C01810=1081.766,322.523,409.402,175.975,26.438,154.460
C01811=1081.760,322.276,409.435,175.972,26.433,154.460
C01812=1081.754,322.027,409.468,175.969,26.429,154.459
C01813=1081.748,321.780,409.500,175.966,26.425,154.458
C01814=1081.742,321.532,409.533,175.963,26.420,154.458
C01815=1081.737,321.283,409.566,175.960,26.416,154.457
C01816=1081.731,321.037,409.598,175.957,26.412,154.457
C01817=1081.725,320.789,409.631,175.954,26.407,154.456
C01818=1081.717,320.468,409.673,175.950,26.402,154.455
C01819=1081.710,320.149,409.715,175.946,26.396,154.454
C01820=1081.702,319.829,409.757,175.943,26.390,154.453
C01821=1081.694,319.509,409.799,175.939,26.385,154.452
C01822=1081.689,319.262,409.831,175.936,26.380,154.452
C01823=1081.684,319.013,409.864,175.933,26.376,154.451
C01824=1081.677,318.766,409.897,175.930,26.372,154.450
C01825=1081.671,318.517,409.929,175.927,26.367,154.450
C01826=1081.666,318.270,409.962,175.924,26.363,154.449
C01827=1081.660,318.022,409.994,175.921,26.359,154.449
C01828=1081.654,317.774,410.026,175.918,26.355,154.448
C01829=1081.648,317.526,410.058,175.915,26.350,154.447
C01830=1081.640,317.181,410.104,175.911,26.344,154.446
C01831=1081.633,316.834,410.149,175.906,26.338,154.445
C01832=1081.625,316.489,410.194,175.903,26.333,154.445
C01833=1081.616,316.143,410.239,175.898,26.326,154.444
C01834=1081.611,315.895,410.271,175.895,26.322,154.443
C01835=1081.605,315.647,410.303,175.892,26.317,154.442
C01836=1081.599,315.399,410.335,175.890,26.314,154.442
C01837=1081.594,315.151,410.368,175.887,26.309,154.441
C01838=1081.588,314.903,410.400,175.884,26.305,154.440
C01839=1081.582,314.655,410.432,175.881,26.301,154.440
C01840=1081.576,314.407,410.464,175.878,26.296,154.439
C01841=1081.570,314.160,410.496,175.875,26.293,154.439
C01842=1081.564,313.912,410.528,175.872,26.288,154.438
C01843=1081.558,313.664,410.560,175.869,26.284,154.437
C01844=1081.552,313.416,410.592,175.866,26.280,154.437
C01845=1081.546,313.168,410.624,175.862,26.276,154.436
C01846=1081.540,312.920,410.656,175.859,26.272,154.436
C01847=1081.534,312.672,410.687,175.857,26.268,154.435
C01848=1081.528,312.424,410.719,175.854,26.264,154.434
C01849=1081.522,312.177,410.751,175.851,26.259,154.434
C01850=1081.516,311.929,410.783,175.848,26.256,154.433
C01851=1081.510,311.681,410.815,175.845,26.251,154.433
C01852=1081.504,311.433,410.847,175.842,26.247,154.432
C01853=1081.498,311.185,410.879,175.839,26.243,154.431
C01854=1081.492,310.937,410.910,175.836,26.239,154.431
C01855=1081.486,310.690,410.942,175.833,26.235,154.430
C01856=1081.480,310.442,410.973,175.831,26.231,154.430
C01857=1081.474,310.194,411.005,175.828,26.227,154.429
C01858=1081.468,309.946,411.037,175.824,26.223,154.428
C01859=1081.463,309.698,411.068,175.821,26.219,154.428
C01860=1081.457,309.450,411.100,175.818,26.215,154.427
C01861=1081.451,309.202,411.131,175.815,26.210,154.427
C01862=1081.445,308.954,411.163,175.812,26.207,154.426
C01863=1081.438,308.706,411.195,175.809,26.202,154.425
C01864=1081.433,308.458,411.227,175.807,26.199,154.425
C01865=1081.427,308.210,411.259,175.804,26.194,154.424
C01866=1081.421,307.962,411.289,175.801,26.190,154.424
C01867=1081.415,307.714,411.321,175.798,26.186,154.423
C01868=1081.410,307.467,411.353,175.795,26.182,154.423
C01869=1081.403,307.219,411.384,175.792,26.178,154.422
C01870=1081.398,306.971,411.416,175.789,26.174,154.421
C01871=1081.392,306.722,411.447,175.787,26.170,154.421
C01872=1081.386,306.475,411.478,175.784,26.166,154.420
C01873=1081.380,306.227,411.510,175.780,26.162,154.420
C01874=1081.375,305.980,411.542,175.777,26.158,154.419
C01875=1081.369,305.732,411.572,175.774,26.154,154.419
C01876=1081.363,305.483,411.604,175.771,26.150,154.418
C01877=1081.357,305.236,411.635,175.768,26.146,154.417
C01878=1081.351,304.987,411.667,175.766,26.142,154.417
C01879=1081.346,304.740,411.698,175.763,26.138,154.416
C01880=1081.339,304.491,411.729,175.760,26.134,154.416
C01881=1081.334,304.244,411.761,175.757,26.130,154.415
C01882=1081.324,303.829,411.813,175.752,26.123,154.414
C01883=1081.314,303.414,411.865,175.747,26.116,154.413
C01884=1081.305,302.999,411.918,175.743,26.109,154.412
C01885=1081.295,302.584,411.970,175.738,26.103,154.411
C01886=1081.289,302.336,412.000,175.735,26.099,154.411
C01887=1081.284,302.088,412.032,175.732,26.095,154.410
C01888=1081.278,301.840,412.063,175.729,26.091,154.409
C01889=1081.272,301.592,412.094,175.726,26.086,154.409
C01890=1081.267,301.344,412.125,175.724,26.083,154.408
C01891=1081.261,301.096,412.156,175.721,26.079,154.408
C01892=1081.255,300.848,412.188,175.718,26.075,154.407
C01893=1081.249,300.600,412.218,175.715,26.071,154.407
C01894=1081.244,300.352,412.249,175.711,26.067,154.406
C01895=1081.238,300.105,412.280,175.709,26.063,154.405
C01896=1081.232,299.856,412.311,175.706,26.059,154.405
C01897=1081.226,299.608,412.342,175.703,26.054,154.404
C01898=1081.221,299.361,412.373,175.700,26.051,154.404
C01899=1081.215,299.113,412.404,175.697,26.047,154.403
C01900=1081.209,298.864,412.435,175.695,26.043,154.402
C01901=1081.203,298.617,412.466,175.692,26.039,154.402
C01902=1081.198,298.369,412.497,175.689,26.035,154.401
C01903=1081.192,298.121,412.528,175.686,26.030,154.401
C01904=1081.187,297.873,412.558,175.684,26.027,154.400
C01905=1081.181,297.624,412.589,175.681,26.023,154.400
C01906=1081.175,297.376,412.620,175.678,26.019,154.399
C01907=1081.170,297.129,412.651,175.674,26.015,154.399
C01908=1081.163,296.880,412.682,175.671,26.011,154.398
C01909=1081.157,296.633,412.712,175.669,26.007,154.397
C01910=1081.152,296.384,412.743,175.666,26.003,154.397
C01911=1081.147,296.137,412.774,175.663,25.999,154.396
C01912=1081.141,295.889,412.804,175.660,25.996,154.396
C01913=1081.134,295.640,412.835,175.658,25.992,154.395
C01914=1081.129,295.392,412.865,175.655,25.988,154.395
C01915=1081.123,295.144,412.896,175.652,25.984,154.394
C01916=1081.118,294.896,412.926,175.649,25.980,154.394
C01917=1081.111,294.648,412.957,175.647,25.976,154.393
C01918=1081.105,294.400,412.987,175.643,25.972,154.393
C01919=1081.100,294.152,413.018,175.640,25.968,154.392
C01920=1081.094,293.904,413.048,175.637,25.965,154.392
C01921=1081.088,293.657,413.078,175.635,25.961,154.391
C01922=1081.082,293.408,413.110,175.632,25.957,154.391
C01923=1081.076,293.160,413.140,175.629,25.953,154.390
C01924=1081.071,292.912,413.170,175.627,25.950,154.389
C01925=1081.065,292.664,413.201,175.624,25.946,154.389
C01926=1081.059,292.417,413.231,175.621,25.942,154.388
C01927=1081.053,292.168,413.261,175.618,25.938,154.388
C01928=1081.047,291.920,413.291,175.615,25.934,154.387
C01929=1081.041,291.672,413.322,175.612,25.930,154.387
C01930=1081.035,291.424,413.352,175.609,25.927,154.386
C01931=1081.030,291.176,413.382,175.606,25.922,154.386
C01932=1081.024,290.928,413.412,175.604,25.919,154.385
C01933=1081.018,290.680,413.442,175.601,25.915,154.385
C01934=1081.009,290.279,413.491,175.596,25.909,154.384
C01935=1081.000,289.878,413.541,175.592,25.902,154.383
C01936=1080.990,289.478,413.589,175.587,25.896,154.382
C01937=1080.981,289.076,413.638,175.583,25.890,154.381
C01938=1080.975,288.829,413.668,175.580,25.886,154.381
C01939=1080.970,288.580,413.698,175.578,25.883,154.380
C01940=1080.964,288.332,413.728,175.574,25.879,154.380
C01941=1080.957,288.084,413.758,175.571,25.875,154.379
C01942=1080.951,287.836,413.788,175.569,25.872,154.379
C01943=1080.946,287.588,413.818,175.566,25.868,154.378
C01944=1080.940,287.339,413.848,175.563,25.864,154.378
C01945=1080.934,287.092,413.878,175.561,25.860,154.377
C01946=1080.929,286.843,413.908,175.558,25.857,154.377
C01947=1080.923,286.595,413.938,175.555,25.853,154.376
C01948=1080.917,286.347,413.967,175.553,25.849,154.376
C01949=1080.911,286.099,413.998,175.549,25.845,154.375
C01950=1080.905,285.851,414.027,175.546,25.842,154.375
C01951=1080.900,285.603,414.058,175.544,25.838,154.374
C01952=1080.894,285.355,414.087,175.541,25.834,154.374
C01953=1080.887,285.107,414.117,175.538,25.830,154.373
C01954=1080.882,284.859,414.147,175.536,25.827,154.373
C01955=1080.876,284.610,414.176,175.533,25.823,154.372
C01956=1080.871,284.362,414.207,175.530,25.819,154.372
C01957=1080.865,284.114,414.236,175.528,25.815,154.371
C01958=1080.859,283.867,414.266,175.524,25.811,154.370
C01959=1080.853,283.618,414.296,175.521,25.808,154.370
C01960=1080.848,283.370,414.325,175.519,25.804,154.370
C01961=1080.842,283.122,414.356,175.516,25.800,154.369
C01962=1080.835,282.874,414.385,175.513,25.797,154.369
C01963=1080.830,282.625,414.414,175.511,25.793,154.368
C01964=1080.824,282.377,414.444,175.508,25.789,154.367
C01965=1080.819,282.129,414.474,175.505,25.785,154.367
C01966=1080.814,281.881,414.503,175.503,25.782,154.366
C01967=1080.807,281.633,414.533,175.499,25.778,154.366
C01968=1080.802,281.385,414.562,175.496,25.774,154.366
C01969=1080.796,281.136,414.592,175.494,25.771,154.365
C01970=1080.790,280.889,414.622,175.491,25.767,154.364
C01971=1080.784,280.640,414.651,175.489,25.763,154.364
C01972=1080.779,280.392,414.681,175.486,25.759,154.363
C01973=1080.773,280.144,414.710,175.483,25.756,154.363
C01974=1080.767,279.895,414.739,175.481,25.752,154.362
C01975=1080.761,279.647,414.769,175.478,25.748,154.362
C01976=1080.755,279.399,414.798,175.474,25.744,154.361
C01977=1080.750,279.151,414.827,175.472,25.741,154.361
C01978=1080.744,278.903,414.856,175.469,25.737,154.361
C01979=1080.739,278.654,414.886,175.467,25.734,154.360
C01980=1080.732,278.406,414.915,175.464,25.730,154.359
C01981=1080.727,278.158,414.945,175.461,25.726,154.359
C01982=1080.721,277.910,414.974,175.459,25.723,154.359
C01983=1080.715,277.661,415.003,175.456,25.719,154.358
C01984=1080.710,277.414,415.032,175.453,25.715,154.357
C01985=1080.704,277.165,415.062,175.450,25.712,154.357
C01986=1080.694,276.775,415.108,175.446,25.706,154.356
C01987=1080.685,276.383,415.154,175.442,25.700,154.356
C01988=1080.676,275.992,415.200,175.437,25.694,154.355
C01989=1080.667,275.601,415.246,175.433,25.689,154.354
C01990=1080.662,275.353,415.274,175.431,25.685,154.353
C01991=1080.656,275.105,415.304,175.428,25.681,154.353
C01992=1080.650,274.857,415.333,175.424,25.678,154.353
C01993=1080.644,274.608,415.362,175.422,25.674,154.352
C01994=1080.638,274.360,415.391,175.419,25.670,154.351
C01995=1080.633,274.112,415.420,175.417,25.666,154.351
C01996=1080.627,273.864,415.449,175.414,25.663,154.351
C01997=1080.621,273.616,415.478,175.411,25.659,154.350
C01998=1080.615,273.367,415.508,175.409,25.655,154.349
C01999=1080.610,273.119,415.536,175.406,25.652,154.349
C02000=1080.604,272.871,415.565,175.404,25.648,154.349
C02001=1080.598,272.623,415.594,175.400,25.645,154.348
C02002=1080.592,272.374,415.623,175.398,25.641,154.348
C02003=1080.587,272.126,415.651,175.395,25.637,154.347
C02004=1080.581,271.878,415.681,175.392,25.634,154.347
C02005=1080.575,271.629,415.709,175.390,25.630,154.346
C02006=1080.569,271.381,415.738,175.387,25.626,154.346
C02007=1080.563,271.134,415.767,175.385,25.623,154.345
C02008=1080.558,270.885,415.796,175.382,25.619,154.345
C02009=1080.552,270.636,415.825,175.379,25.616,154.344
C02010=1080.547,270.388,415.853,175.376,25.612,154.344
C02011=1080.540,270.140,415.882,175.374,25.609,154.343
C02012=1080.535,269.891,415.911,175.371,25.605,154.343
C02013=1080.529,269.643,415.940,175.368,25.601,154.342
C02014=1080.523,269.395,415.968,175.366,25.598,154.342
C02015=1080.517,269.147,415.997,175.363,25.594,154.341
C02016=1080.511,268.898,416.025,175.361,25.591,154.341
C02017=1080.506,268.651,416.054,175.357,25.587,154.340
C02018=1080.500,268.402,416.083,175.355,25.584,154.340
C02019=1080.494,268.153,416.112,175.352,25.580,154.340
C02020=1080.489,267.905,416.140,175.350,25.576,154.339
C02021=1080.483,267.657,416.168,175.347,25.573,154.339
C02022=1080.477,267.409,416.197,175.345,25.569,154.338
C02023=1080.471,267.161,416.225,175.342,25.566,154.338
C02024=1080.465,266.912,416.254,175.339,25.562,154.337
C02025=1080.460,266.664,416.282,175.336,25.558,154.337
C02026=1080.455,266.415,416.311,175.333,25.555,154.336
C02027=1080.448,266.167,416.340,175.331,25.551,154.336
C02028=1080.443,265.919,416.368,175.328,25.548,154.335
C02029=1080.437,265.670,416.396,175.326,25.544,154.335
C02030=1080.431,265.422,416.425,175.323,25.540,154.334
C02031=1080.425,265.174,416.453,175.321,25.537,154.334
C02032=1080.419,264.925,416.482,175.318,25.533,154.333
C02033=1080.414,264.677,416.510,175.315,25.530,154.333
C02034=1080.408,264.429,416.538,175.312,25.526,154.332
C02035=1080.403,264.181,416.567,175.310,25.522,154.332
C02036=1080.397,263.932,416.595,175.307,25.519,154.331
C02037=1080.391,263.684,416.623,175.305,25.515,154.331
C02038=1080.382,263.296,416.667,175.300,25.510,154.330
C02039=1080.373,262.908,416.712,175.297,25.505,154.330
C02040=1080.363,262.520,416.756,175.292,25.499,154.329
C02041=1080.354,262.132,416.799,175.288,25.494,154.328
C02042=1080.348,261.884,416.827,175.285,25.490,154.328
C02043=1080.342,261.636,416.856,175.283,25.487,154.327
C02044=1080.336,261.387,416.884,175.280,25.483,154.327
C02045=1080.330,261.139,416.911,175.278,25.480,154.326
C02046=1080.324,260.890,416.940,175.275,25.476,154.326
C02047=1080.319,260.642,416.968,175.272,25.473,154.325
C02048=1080.313,260.394,416.996,175.269,25.469,154.325
C02049=1080.307,260.146,417.023,175.267,25.465,154.325
C02050=1080.301,259.897,417.052,175.264,25.462,154.324
C02051=1080.296,259.648,417.079,175.262,25.458,154.324
C02052=1080.290,259.400,417.107,175.259,25.455,154.323
C02053=1080.284,259.152,417.135,175.257,25.452,154.323
C02054=1080.278,258.903,417.163,175.254,25.448,154.322
C02055=1080.272,258.655,417.191,175.251,25.445,154.322
C02056=1080.267,258.406,417.219,175.248,25.441,154.321
C02057=1080.260,258.159,417.247,175.246,25.438,154.321
C02058=1080.255,257.910,417.275,175.243,25.434,154.320
C02059=1080.249,257.662,417.303,175.241,25.431,154.320
C02060=1080.243,257.413,417.330,175.238,25.427,154.320
C02061=1080.237,257.165,417.358,175.236,25.423,154.319
C02062=1080.232,256.916,417.386,175.233,25.420,154.319
C02063=1080.226,256.668,417.414,175.230,25.416,154.318
C02064=1080.220,256.420,417.441,175.228,25.413,154.318
C02065=1080.214,256.171,417.469,175.225,25.409,154.317
C02066=1080.209,255.923,417.497,175.223,25.406,154.317
C02067=1080.202,255.674,417.525,175.220,25.402,154.316
C02068=1080.197,255.426,417.552,175.218,25.399,154.316
C02069=1080.191,255.177,417.580,175.215,25.395,154.315
C02070=1080.185,254.929,417.608,175.212,25.392,154.315
C02071=1080.180,254.681,417.636,175.209,25.388,154.315
C02072=1080.174,254.432,417.663,175.207,25.385,154.314
C02073=1080.168,254.184,417.691,175.205,25.381,154.314
C02074=1080.163,253.935,417.718,175.202,25.378,154.313
C02075=1080.157,253.687,417.746,175.200,25.374,154.313
C02076=1080.151,253.439,417.774,175.197,25.371,154.312
C02077=1080.146,253.190,417.801,175.195,25.367,154.312
C02078=1080.140,252.942,417.829,175.191,25.364,154.311
C02079=1080.134,252.693,417.856,175.189,25.360,154.311
C02080=1080.129,252.445,417.884,175.186,25.356,154.311
C02081=1080.122,252.196,417.911,175.184,25.353,154.310
C02082=1080.117,251.948,417.939,175.182,25.350,154.310
C02083=1080.111,251.700,417.966,175.179,25.346,154.309
C02084=1080.106,251.451,417.994,175.177,25.343,154.309
C02085=1080.100,251.203,418.022,175.174,25.339,154.308
C02086=1080.095,250.954,418.048,175.172,25.335,154.308
C02087=1080.089,250.706,418.076,175.168,25.332,154.307
C02088=1080.083,250.457,418.103,175.166,25.328,154.307
C02089=1080.078,250.209,418.131,175.164,25.325,154.306
C02090=1080.069,249.818,418.174,175.159,25.319,154.306
C02091=1080.060,249.427,418.217,175.156,25.314,154.305
C02092=1080.051,249.037,418.259,175.152,25.308,154.304
C02093=1080.042,248.646,418.303,175.148,25.302,154.303
C02094=1080.037,248.397,418.330,175.146,25.299,154.303
C02095=1080.031,248.149,418.357,175.143,25.295,154.302
C02096=1080.025,247.901,418.385,175.140,25.292,154.302
C02097=1080.020,247.652,418.412,175.138,25.288,154.301
C02098=1080.014,247.403,418.439,175.135,25.285,154.301
C02099=1080.009,247.155,418.467,175.133,25.281,154.301
C02100=1080.003,246.907,418.494,175.130,25.278,154.300
C02101=1079.997,246.658,418.520,175.128,25.274,154.300
C02102=1079.992,246.410,418.547,175.126,25.271,154.299
C02103=1079.986,246.161,418.574,175.123,25.267,154.299
C02104=1079.980,245.913,418.602,175.120,25.264,154.298
C02105=1079.975,245.664,418.629,175.117,25.260,154.298
C02106=1079.969,245.416,418.656,175.115,25.257,154.297
C02107=1079.963,245.168,418.682,175.113,25.253,154.297
C02108=1079.957,244.918,418.710,175.110,25.249,154.296
C02109=1079.952,244.670,418.737,175.108,25.246,154.296
C02110=1079.946,244.422,418.764,175.105,25.242,154.296
C02111=1079.941,244.173,418.791,175.103,25.239,154.295
C02112=1079.935,243.925,418.818,175.100,25.236,154.295
C02113=1079.929,243.677,418.845,175.097,25.232,154.294
C02114=1079.924,243.428,418.872,175.095,25.228,154.294
C02115=1079.918,243.179,418.899,175.093,25.225,154.293
C02116=1079.912,242.931,418.925,175.090,25.221,154.293
C02117=1079.906,242.682,418.952,175.088,25.218,154.292
C02118=1079.901,242.434,418.979,175.086,25.215,154.292
C02119=1079.895,242.185,419.006,175.083,25.211,154.291
C02120=1079.889,241.937,419.033,175.080,25.208,154.291
C02121=1079.884,241.689,419.059,175.077,25.204,154.291
C02122=1079.877,241.439,419.086,175.075,25.201,154.290
C02123=1079.872,241.191,419.113,175.073,25.198,154.290
C02124=1079.866,240.943,419.140,175.070,25.194,154.289
C02125=1079.860,240.694,419.166,175.068,25.190,154.289
C02126=1079.854,240.446,419.193,175.066,25.187,154.288
C02127=1079.849,240.197,419.220,175.063,25.183,154.288
C02128=1079.844,239.948,419.246,175.060,25.180,154.288
C02129=1079.838,239.700,419.273,175.058,25.177,154.287
C02130=1079.832,239.452,419.299,175.055,25.173,154.287
C02131=1079.826,239.203,419.326,175.053,25.170,154.286
C02132=1079.820,238.954,419.353,175.051,25.166,154.286
C02133=1079.814,238.706,419.380,175.048,25.163,154.285
C02134=1079.809,238.457,419.406,175.046,25.159,154.285
C02135=1079.803,238.209,419.432,175.043,25.156,154.284
C02136=1079.797,237.960,419.459,175.040,25.152,154.284
C02137=1079.791,237.712,419.486,175.038,25.149,154.283
C02138=1079.786,237.463,419.511,175.035,25.145,154.283
C02139=1079.780,237.214,419.538,175.033,25.142,154.283
C02140=1079.774,236.966,419.565,175.031,25.138,154.282
C02141=1079.769,236.718,419.591,175.028,25.135,154.282
C02142=1079.760,236.320,419.633,175.024,25.130,154.281
C02143=1079.750,235.922,419.676,175.021,25.124,154.280
C02144=1079.741,235.525,419.719,175.017,25.119,154.280
C02145=1079.732,235.128,419.760,175.013,25.112,154.279
C02146=1079.726,234.880,419.786,175.010,25.109,154.278
C02147=1079.721,234.631,419.812,175.008,25.106,154.278
C02148=1079.715,234.382,419.839,175.005,25.102,154.277
C02149=1079.710,234.133,419.865,175.003,25.099,154.277
C02150=1079.704,233.885,419.891,175.001,25.095,154.277
C02151=1079.698,233.637,419.918,174.998,25.092,154.276
C02152=1079.693,233.388,419.944,174.996,25.088,154.276
C02153=1079.687,233.139,419.971,174.994,25.085,154.275
C02154=1079.681,232.890,419.997,174.991,25.082,154.275
C02155=1079.676,232.642,420.023,174.988,25.078,154.274
C02156=1079.669,232.393,420.049,174.986,25.075,154.274
C02157=1079.664,232.145,420.075,174.984,25.072,154.274
C02158=1079.658,231.896,420.101,174.981,25.068,154.273
C02159=1079.653,231.647,420.127,174.979,25.064,154.273
C02160=1079.647,231.399,420.154,174.977,25.061,154.272
C02161=1079.642,231.150,420.179,174.974,25.057,154.272
C02162=1079.636,230.902,420.205,174.972,25.054,154.271
C02163=1079.630,230.653,420.231,174.970,25.050,154.271
C02164=1079.624,230.405,420.258,174.966,25.047,154.270
C02165=1079.619,230.156,420.284,174.964,25.043,154.270
C02166=1079.613,229.907,420.309,174.962,25.040,154.269
C02167=1079.607,229.659,420.336,174.960,25.037,154.269
C02168=1079.601,229.410,420.362,174.957,25.033,154.269
C02169=1079.595,229.161,420.387,174.955,25.030,154.268
C02170=1079.589,228.913,420.414,174.953,25.027,154.268
C02171=1079.585,228.665,420.439,174.951,25.023,154.267
C02172=1079.578,228.416,420.465,174.947,25.019,154.267
C02173=1079.573,228.167,420.491,174.945,25.016,154.266
C02174=1079.566,227.919,420.517,174.943,25.013,154.266
C02175=1079.561,227.670,420.543,174.940,25.009,154.266
C02176=1079.555,227.421,420.568,174.938,25.006,154.265
C02177=1079.549,227.172,420.594,174.936,25.002,154.265
C02178=1079.543,226.924,420.620,174.934,24.999,154.264
C02179=1079.539,226.676,420.646,174.931,24.995,154.264
C02180=1079.532,226.427,420.671,174.929,24.992,154.263
C02181=1079.527,226.178,420.697,174.926,24.989,154.263
C02182=1079.521,225.929,420.723,174.924,24.985,154.262
C02183=1079.515,225.680,420.749,174.921,24.982,154.262
C02184=1079.509,225.433,420.774,174.919,24.978,154.262
C02185=1079.504,225.184,420.800,174.917,24.975,154.261
C02186=1079.498,224.935,420.826,174.915,24.972,154.261
C02187=1079.492,224.686,420.851,174.912,24.968,154.260
C02188=1079.487,224.437,420.877,174.910,24.964,154.260
C02189=1079.481,224.189,420.902,174.907,24.961,154.259
C02190=1079.476,223.940,420.928,174.905,24.958,154.259
C02191=1079.469,223.692,420.954,174.902,24.954,154.258
C02192=1079.464,223.443,420.980,174.900,24.950,154.258
C02193=1079.458,223.195,421.005,174.898,24.947,154.258
C02194=1079.450,222.789,421.047,174.895,24.942,154.257
C02195=1079.440,222.382,421.089,174.890,24.935,154.256
C02196=1079.431,221.977,421.130,174.887,24.930,154.255
C02197=1079.422,221.571,421.172,174.883,24.925,154.255
C02198=1079.415,221.322,421.197,174.880,24.921,154.254
C02199=1079.410,221.073,421.223,174.878,24.917,154.254
C02200=1079.404,220.825,421.248,174.876,24.914,154.253
C02201=1079.398,220.577,421.273,174.874,24.911,154.253
C02202=1079.393,220.327,421.298,174.871,24.907,154.252
C02203=1079.387,220.079,421.324,174.868,24.904,154.252
C02204=1079.381,219.831,421.349,174.866,24.901,154.252
C02205=1079.376,219.582,421.375,174.864,24.897,154.251
C02206=1079.370,219.333,421.400,174.862,24.894,154.251
C02207=1079.363,219.084,421.425,174.859,24.890,154.250
C02208=1079.359,218.835,421.450,174.857,24.887,154.250
C02209=1079.353,218.587,421.476,174.855,24.883,154.249
C02210=1079.346,218.338,421.501,174.853,24.880,154.249
C02211=1079.341,218.090,421.526,174.851,24.877,154.248
C02212=1079.336,217.840,421.551,174.847,24.873,154.248
C02213=1079.329,217.592,421.576,174.845,24.869,154.247
C02214=1079.324,217.344,421.601,174.843,24.866,154.247
C02215=1079.318,217.095,421.627,174.841,24.863,154.247
C02216=1079.313,216.846,421.652,174.839,24.859,154.246
C02217=1079.307,216.598,421.677,174.836,24.856,154.246
C02218=1079.301,216.349,421.702,174.834,24.853,154.245
C02219=1079.296,216.100,421.727,174.832,24.849,154.245
C02220=1079.290,215.851,421.752,174.830,24.846,154.244
C02221=1079.284,215.603,421.778,174.828,24.842,154.244
C02222=1079.278,215.354,421.802,174.824,24.839,154.244
C02223=1079.273,215.105,421.828,174.822,24.835,154.243
C02224=1079.267,214.857,421.853,174.820,24.832,154.243
C02225=1079.261,214.608,421.878,174.818,24.828,154.242
C02226=1079.256,214.360,421.903,174.816,24.825,154.242
C02227=1079.250,214.111,421.927,174.813,24.821,154.241
C02228=1079.244,213.862,421.953,174.811,24.818,154.241
C02229=1079.239,213.613,421.977,174.809,24.814,154.240
C02230=1079.233,213.364,422.003,174.807,24.811,154.240
C02231=1079.228,213.116,422.027,174.805,24.807,154.239
C02232=1079.221,212.867,422.052,174.802,24.804,154.239
C02233=1079.216,212.619,422.077,174.799,24.800,154.239
C02234=1079.211,212.370,422.103,174.797,24.797,154.238
C02235=1079.205,212.121,422.127,174.795,24.794,154.238
C02236=1079.199,211.872,422.152,174.793,24.790,154.237
C02237=1079.194,211.624,422.176,174.791,24.787,154.237
C02238=1079.188,211.375,422.202,174.789,24.783,154.236
C02239=1079.182,211.126,422.226,174.786,24.780,154.236
C02240=1079.176,210.878,422.251,174.784,24.777,154.236
C02241=1079.170,210.628,422.276,174.782,24.773,154.235
C02242=1079.165,210.380,422.300,174.780,24.770,154.235
C02243=1079.159,210.131,422.326,174.777,24.766,154.234
C02244=1079.153,209.883,422.350,174.775,24.763,154.234
C02245=1079.147,209.633,422.374,174.772,24.759,154.233
C02246=1079.138,209.232,422.415,174.769,24.753,154.232
C02247=1079.129,208.830,422.455,174.765,24.748,154.232
C02248=1079.120,208.428,422.494,174.762,24.742,154.231
C02249=1079.111,208.027,422.534,174.758,24.737,154.230
C02250=1079.087,206.992,422.634,174.654,24.681,154.232
C02251=1079.082,206.742,422.658,174.651,24.679,154.231
C02252=1079.076,206.494,422.682,174.649,24.677,154.231
C02253=1079.071,206.245,422.706,174.647,24.674,154.231
C02254=1079.065,205.997,422.730,174.644,24.672,154.231
C02255=1079.059,205.749,422.754,174.642,24.669,154.231
C02256=1079.054,205.499,422.778,174.640,24.666,154.230
C02257=1079.048,205.250,422.802,174.637,24.664,154.230
C02258=1079.042,205.002,422.826,174.635,24.662,154.230
C02259=1079.037,204.753,422.850,174.633,24.659,154.230
C02260=1079.031,204.503,422.874,174.630,24.657,154.229
C02261=1079.025,204.255,422.897,174.628,24.654,154.229
C02262=1079.020,204.006,422.922,174.625,24.651,154.229
C02263=1079.015,203.757,422.945,174.623,24.649,154.229
C02264=1079.009,203.509,422.969,174.621,24.647,154.228
C02265=1079.004,203.260,422.993,174.618,24.644,154.228
C02266=1078.998,203.010,423.017,174.616,24.642,154.228
C02267=1078.992,202.762,423.041,174.614,24.639,154.228
C02268=1078.987,202.514,423.065,174.611,24.637,154.228
C02269=1078.981,202.265,423.088,174.609,24.634,154.227
C02270=1078.976,202.016,423.112,174.607,24.632,154.227
C02271=1078.969,201.767,423.136,174.604,24.630,154.227
C02272=1078.963,201.518,423.159,174.602,24.627,154.227
C02273=1078.958,201.270,423.183,174.599,24.625,154.227
C02274=1078.952,201.021,423.206,174.597,24.622,154.226
C02275=1078.947,200.772,423.231,174.595,24.620,154.226
C02276=1078.941,200.523,423.254,174.592,24.617,154.226
C02277=1078.935,200.274,423.278,174.590,24.615,154.226
C02278=1078.930,200.025,423.301,174.588,24.612,154.225
C02279=1078.924,199.777,423.325,174.585,24.610,154.225
C02280=1078.919,199.528,423.348,174.583,24.608,154.225
C02281=1078.913,199.279,423.372,174.580,24.605,154.225
C02282=1078.907,199.030,423.395,174.578,24.603,154.225
C02283=1078.901,198.781,423.420,174.576,24.601,154.225
C02284=1078.895,198.532,423.443,174.573,24.598,154.224
C02285=1078.890,198.284,423.467,174.572,24.596,154.224
C02286=1078.884,198.035,423.490,174.570,24.594,154.224
C02287=1078.878,197.786,423.513,174.567,24.591,154.224
C02288=1078.873,197.537,423.537,174.565,24.589,154.223
C02289=1078.867,197.288,423.560,174.563,24.586,154.223
C02290=1078.861,197.040,423.584,174.560,24.584,154.223
C02291=1078.856,196.791,423.607,174.558,24.581,154.223
C02292=1078.850,196.542,423.631,174.555,24.579,154.223
C02293=1078.844,196.293,423.654,174.553,24.576,154.222
C02294=1078.839,196.044,423.678,174.551,24.574,154.222
C02295=1078.833,195.796,423.701,174.548,24.572,154.222
C02296=1078.827,195.547,423.724,174.546,24.569,154.222
C02297=1078.822,195.297,423.748,174.544,24.567,154.221
C02298=1078.817,195.049,423.771,174.541,24.564,154.221
C02299=1078.811,194.800,423.794,174.539,24.562,154.221
C02300=1078.806,194.551,423.818,174.537,24.559,154.221
C02301=1078.800,194.302,423.841,174.534,24.557,154.221
C02302=1078.794,194.054,423.865,174.533,24.555,154.220
C02303=1078.788,193.805,423.887,174.531,24.552,154.220
C02304=1078.783,193.556,423.911,174.528,24.550,154.220
C02305=1078.777,193.307,423.934,174.526,24.547,154.220
C02306=1078.772,193.058,423.957,174.523,24.545,154.220
C02307=1078.766,192.809,423.981,174.521,24.542,154.219
C02308=1078.761,192.561,424.004,174.519,24.540,154.219
C02309=1078.755,192.312,424.027,174.516,24.538,154.219
C02310=1078.749,192.063,424.050,174.514,24.535,154.219
C02311=1078.743,191.782,424.077,174.512,24.532,154.218
C02312=1078.737,191.503,424.102,174.509,24.530,154.218
C02313=1078.730,191.223,424.129,174.506,24.526,154.218
C02314=1078.724,190.942,424.155,174.504,24.524,154.218
C02315=1078.718,190.693,424.178,174.501,24.522,154.217
C02316=1078.713,190.445,424.201,174.499,24.519,154.217
C02317=1078.708,190.196,424.224,174.498,24.517,154.217
C02318=1078.703,189.947,424.247,174.495,24.514,154.217
C02319=1078.697,189.698,424.270,174.493,24.512,154.216
C02320=1078.691,189.449,424.293,174.491,24.510,154.216
C02321=1078.685,189.200,424.316,174.488,24.507,154.216
C02322=1078.680,188.951,424.340,174.486,24.504,154.216
C02323=1078.675,188.702,424.363,174.484,24.502,154.216
C02324=1078.669,188.453,424.386,174.481,24.499,154.215
C02325=1078.663,188.205,424.409,174.479,24.497,154.215
C02326=1078.658,187.956,424.431,174.478,24.495,154.215
C02327=1078.653,187.707,424.455,174.475,24.492,154.215
C02328=1078.647,187.458,424.478,174.473,24.490,154.215
C02329=1078.642,187.209,424.501,174.471,24.487,154.214
C02330=1078.636,186.960,424.524,174.468,24.485,154.214
C02331=1078.630,186.712,424.546,174.466,24.483,154.214
C02332=1078.625,186.462,424.570,174.464,24.480,154.214
C02333=1078.620,186.214,424.593,174.462,24.478,154.213
C02334=1078.614,185.965,424.616,174.460,24.475,154.213
C02335=1078.609,185.716,424.638,174.457,24.473,154.213
C02336=1078.603,185.467,424.661,174.455,24.470,154.213
C02337=1078.597,185.218,424.684,174.453,24.468,154.212
C02338=1078.593,184.969,424.707,174.450,24.465,154.212
C02339=1078.587,184.721,424.729,174.448,24.463,154.212
C02340=1078.581,184.472,424.752,174.447,24.461,154.212
C02341=1078.575,184.223,424.775,174.444,24.459,154.212
C02342=1078.570,183.974,424.797,174.442,24.456,154.211
C02343=1078.564,183.725,424.820,174.439,24.454,154.211
C02344=1078.558,183.476,424.843,174.437,24.452,154.211
C02345=1078.552,183.227,424.866,174.435,24.449,154.211
C02346=1078.546,182.978,424.888,174.433,24.447,154.211
C02347=1078.541,182.729,424.911,174.431,24.444,154.210
C02348=1078.534,182.480,424.933,174.428,24.442,154.210
C02349=1078.528,182.231,424.956,174.426,24.440,154.210
C02350=1078.524,181.982,424.978,174.424,24.437,154.210
C02351=1078.518,181.734,425.001,174.421,24.435,154.210
C02352=1078.511,181.485,425.023,174.420,24.433,154.209
C02353=1078.506,181.236,425.046,174.418,24.431,154.209
C02354=1078.500,180.987,425.068,174.415,24.428,154.209
C02355=1078.495,180.738,425.091,174.413,24.426,154.209
C02356=1078.488,180.489,425.114,174.411,24.423,154.209
C02357=1078.483,180.240,425.135,174.409,24.421,154.208
C02358=1078.477,179.991,425.158,174.407,24.419,154.208
C02359=1078.472,179.742,425.181,174.404,24.417,154.208
C02360=1078.466,179.493,425.203,174.402,24.414,154.208
C02361=1078.460,179.244,425.226,174.400,24.412,154.208
C02362=1078.454,178.995,425.248,174.398,24.409,154.207
C02363=1078.449,178.747,425.271,174.396,24.407,154.207
C02364=1078.443,178.498,425.293,174.394,24.405,154.207
C02365=1078.437,178.249,425.315,174.391,24.402,154.207
C02366=1078.432,178.000,425.338,174.389,24.400,154.206
C02367=1078.426,177.750,425.360,174.387,24.398,154.206
C02368=1078.420,177.502,425.383,174.385,24.395,154.206
C02369=1078.415,177.253,425.405,174.383,24.393,154.206
C02370=1078.408,177.004,425.427,174.380,24.390,154.206
C02371=1078.403,176.755,425.449,174.378,24.388,154.206
C02372=1078.398,176.506,425.472,174.376,24.386,154.205
C02373=1078.393,176.257,425.494,174.374,24.384,154.205
C02374=1078.386,176.008,425.516,174.372,24.381,154.205
C02375=1078.380,175.728,425.542,174.369,24.379,154.205
C02376=1078.374,175.448,425.567,174.367,24.376,154.204
C02377=1078.367,175.167,425.592,174.365,24.373,154.204
C02378=1078.361,174.886,425.616,174.363,24.371,154.204
C02379=1078.355,174.638,425.639,174.360,24.369,154.204
C02380=1078.349,174.388,425.661,174.358,24.366,154.203
C02381=1078.344,174.140,425.683,174.356,24.363,154.203
C02382=1078.339,173.891,425.706,174.353,24.361,154.203
C02383=1078.332,173.641,425.727,174.352,24.359,154.203
C02384=1078.327,173.393,425.750,174.349,24.357,154.203
C02385=1078.322,173.144,425.772,174.347,24.354,154.202
C02386=1078.316,172.895,425.794,174.345,24.352,154.202
C02387=1078.311,172.646,425.816,174.343,24.349,154.202
C02388=1078.305,172.397,425.838,174.341,24.347,154.202
C02389=1078.299,172.148,425.860,174.339,24.344,154.202
C02390=1078.294,171.899,425.883,174.336,24.342,154.201
C02391=1078.288,171.650,425.904,174.335,24.340,154.201
C02392=1078.283,171.401,425.926,174.332,24.337,154.201
C02393=1078.277,171.152,425.949,174.330,24.335,154.201
C02394=1078.271,170.903,425.971,174.328,24.332,154.200
C02395=1078.266,170.654,425.993,174.326,24.330,154.200
C02396=1078.260,170.405,426.014,174.324,24.328,154.200
C02397=1078.254,170.156,426.037,174.322,24.325,154.200
C02398=1078.249,169.908,426.059,174.320,24.323,154.200
C02399=1078.243,169.658,426.081,174.318,24.321,154.199
C02400=1078.238,169.410,426.102,174.316,24.318,154.199
C02401=1078.232,169.160,426.124,174.313,24.316,154.199
C02402=1078.227,168.912,426.147,174.312,24.314,154.199
C02403=1078.221,168.663,426.168,174.309,24.311,154.198
C02404=1078.216,168.413,426.191,174.307,24.309,154.198
C02405=1078.211,168.165,426.212,174.305,24.306,154.198
C02406=1078.205,167.915,426.234,174.303,24.304,154.198
C02407=1078.200,167.667,426.256,174.301,24.301,154.197
C02408=1078.194,167.417,426.278,174.299,24.299,154.197
C02409=1078.188,167.169,426.300,174.297,24.297,154.197
C02410=1078.182,166.920,426.322,174.295,24.294,154.197
C02411=1078.177,166.671,426.344,174.293,24.292,154.197
C02412=1078.171,166.422,426.365,174.290,24.289,154.196
C02413=1078.167,166.173,426.387,174.289,24.287,154.196
C02414=1078.160,165.924,426.409,174.287,24.285,154.196
C02415=1078.156,165.675,426.431,174.284,24.282,154.196
C02416=1078.149,165.426,426.452,174.283,24.280,154.195
C02417=1078.145,165.177,426.474,174.281,24.278,154.195
C02418=1078.139,164.928,426.496,174.278,24.275,154.195
C02419=1078.134,164.679,426.518,174.277,24.273,154.195
C02420=1078.128,164.430,426.540,174.274,24.270,154.195
C02421=1078.123,164.181,426.561,174.272,24.268,154.194
C02422=1078.117,163.932,426.583,174.271,24.265,154.194
C02423=1078.112,163.683,426.605,174.269,24.263,154.194
C02424=1078.106,163.434,426.627,174.266,24.260,154.194
C02425=1078.101,163.185,426.648,174.264,24.258,154.193
C02426=1078.095,162.935,426.670,174.263,24.255,154.193
C02427=1078.090,162.687,426.692,174.260,24.253,154.193
C02428=1078.084,162.438,426.713,174.258,24.251,154.193
C02429=1078.079,162.189,426.735,174.256,24.248,154.192
C02430=1078.073,161.940,426.756,174.254,24.246,154.192
C02431=1078.068,161.690,426.778,174.252,24.243,154.192
C02432=1078.062,161.442,426.799,174.250,24.241,154.192
C02433=1078.057,161.192,426.821,174.248,24.239,154.192
C02434=1078.051,160.944,426.843,174.246,24.236,154.191
C02435=1078.045,160.695,426.864,174.244,24.234,154.191
C02436=1078.040,160.446,426.886,174.242,24.232,154.191
C02437=1078.034,160.197,426.907,174.240,24.229,154.191
C02438=1078.029,159.947,426.928,174.238,24.227,154.190
C02439=1078.022,159.666,426.952,174.236,24.224,154.190
C02440=1078.016,159.386,426.976,174.234,24.222,154.190
C02441=1078.009,159.105,427.000,174.231,24.219,154.190
C02442=1078.003,158.824,427.025,174.229,24.216,154.189
C02443=1077.998,158.576,427.046,174.227,24.214,154.189
C02444=1077.992,158.327,427.068,174.224,24.211,154.189
C02445=1077.986,158.078,427.089,174.223,24.209,154.189
C02446=1077.980,157.828,427.110,174.221,24.207,154.189
C02447=1077.975,157.579,427.132,174.218,24.204,154.188
C02448=1077.969,157.330,427.153,174.217,24.202,154.188
C02449=1077.964,157.082,427.175,174.215,24.200,154.188
C02450=1077.958,156.833,427.195,174.213,24.197,154.188
C02451=1077.952,156.583,427.217,174.211,24.195,154.187
C02452=1077.947,156.335,427.238,174.209,24.192,154.187
C02453=1077.941,156.085,427.259,174.207,24.190,154.187
C02454=1077.936,155.836,427.281,174.205,24.188,154.187
C02455=1077.931,155.588,427.302,174.203,24.185,154.186
C02456=1077.925,155.338,427.323,174.201,24.183,154.186
C02457=1077.919,155.089,427.344,174.199,24.181,154.186
C02458=1077.913,154.840,427.365,174.197,24.178,154.186
C02459=1077.908,154.591,427.386,174.195,24.176,154.186
C02460=1077.902,154.343,427.408,174.193,24.173,154.185
C02461=1077.896,154.093,427.429,174.191,24.172,154.185
C02462=1077.891,153.844,427.450,174.189,24.169,154.185
C02463=1077.885,153.594,427.471,174.187,24.167,154.185
C02464=1077.879,153.346,427.492,174.185,24.164,154.184
C02465=1077.874,153.097,427.513,174.183,24.162,154.184
C02466=1077.868,152.848,427.534,174.181,24.159,154.184
C02467=1077.863,152.599,427.555,174.179,24.157,154.184
C02468=1077.857,152.350,427.576,174.177,24.154,154.183
C02469=1077.851,152.100,427.597,174.175,24.153,154.183
C02470=1077.846,151.852,427.618,174.173,24.150,154.183
C02471=1077.840,151.603,427.639,174.171,24.148,154.183
C02472=1077.834,151.353,427.660,174.169,24.145,154.183
C02473=1077.829,151.104,427.681,174.167,24.143,154.182
C02474=1077.823,150.856,427.702,174.166,24.141,154.182
C02475=1077.818,150.606,427.723,174.163,24.138,154.182
C02476=1077.812,150.357,427.744,174.161,24.135,154.182
C02477=1077.807,150.108,427.765,174.160,24.134,154.181
C02478=1077.801,149.859,427.787,174.157,24.131,154.181
C02479=1077.795,149.610,427.807,174.156,24.129,154.181
C02480=1077.789,149.361,427.827,174.154,24.126,154.181
C02481=1077.784,149.113,427.848,174.151,24.124,154.181
C02482=1077.778,148.863,427.869,174.150,24.121,154.180
C02483=1077.772,148.614,427.891,174.148,24.119,154.180
C02484=1077.767,148.365,427.911,174.146,24.117,154.180
C02485=1077.761,148.115,427.932,174.144,24.115,154.180
C02486=1077.756,147.867,427.953,174.142,24.112,154.179
C02487=1077.750,147.618,427.974,174.140,24.109,154.179
C02488=1077.744,147.369,427.994,174.138,24.107,154.179
C02489=1077.739,147.119,428.015,174.136,24.105,154.179
C02490=1077.733,146.871,428.036,174.134,24.103,154.179
C02491=1077.728,146.621,428.057,174.133,24.100,154.178
C02492=1077.721,146.372,428.077,174.130,24.098,154.178
C02493=1077.716,146.123,428.098,174.128,24.095,154.178
C02494=1077.710,145.874,428.119,174.127,24.093,154.178
C02495=1077.705,145.625,428.139,174.124,24.090,154.177
C02496=1077.698,145.376,428.160,174.123,24.089,154.177
C02497=1077.693,145.127,428.181,174.121,24.086,154.177
C02498=1077.688,144.878,428.201,174.119,24.084,154.177
C02499=1077.682,144.629,428.222,174.117,24.081,154.176
C02500=1077.676,144.379,428.242,174.115,24.079,154.176
C02501=1077.671,144.130,428.263,174.113,24.077,154.176
C02502=1077.665,143.882,428.284,174.111,24.074,154.176
C02503=1077.659,143.601,428.307,174.109,24.071,154.175
C02504=1077.652,143.319,428.331,174.107,24.069,154.175
C02505=1077.646,143.038,428.353,174.105,24.066,154.175
C02506=1077.639,142.758,428.377,174.103,24.064,154.175
C02507=1077.634,142.508,428.398,174.101,24.061,154.174
C02508=1077.628,142.259,428.418,174.099,24.059,154.174
C02509=1077.622,142.010,428.438,174.097,24.056,154.174
C02510=1077.617,141.761,428.459,174.095,24.054,154.174
C02511=1077.612,141.512,428.479,174.093,24.051,154.173
C02512=1077.607,141.263,428.500,174.091,24.049,154.173
C02513=1077.600,141.013,428.520,174.089,24.047,154.173
C02514=1077.595,140.764,428.541,174.087,24.044,154.173
C02515=1077.589,140.515,428.561,174.086,24.042,154.173
C02516=1077.583,140.266,428.581,174.083,24.039,154.172
C02517=1077.578,140.017,428.602,174.082,24.037,154.172
C02518=1077.572,139.768,428.622,174.080,24.035,154.172
C02519=1077.566,139.519,428.643,174.078,24.033,154.172
C02520=1077.561,139.270,428.664,174.076,24.030,154.171
C02521=1077.555,139.021,428.684,174.075,24.028,154.171
C02522=1077.550,138.772,428.704,174.072,24.025,154.171
C02523=1077.544,138.523,428.724,174.071,24.023,154.171
C02524=1077.539,138.274,428.744,174.069,24.020,154.170
C02525=1077.532,138.024,428.765,174.066,24.018,154.170
C02526=1077.527,137.775,428.785,174.065,24.016,154.170
C02527=1077.521,137.526,428.805,174.063,24.013,154.170
C02528=1077.516,137.277,428.826,174.061,24.011,154.169
C02529=1077.510,137.028,428.846,174.059,24.008,154.169
C02530=1077.504,136.779,428.866,174.058,24.006,154.169
C02531=1077.498,136.530,428.886,174.055,24.004,154.169
C02532=1077.492,136.280,428.907,174.054,24.001,154.168
C02533=1077.486,136.032,428.927,174.052,23.999,154.168
C02534=1077.481,135.783,428.948,174.050,23.997,154.168
C02535=1077.475,135.533,428.967,174.048,23.994,154.168
C02536=1077.470,135.284,428.987,174.047,23.992,154.168
C02537=1077.464,135.035,429.007,174.044,23.989,154.167
C02538=1077.459,134.786,429.028,174.043,23.987,154.167
C02539=1077.453,134.537,429.048,174.041,23.985,154.167
C02540=1077.448,134.288,429.068,174.039,23.982,154.167
C02541=1077.442,134.039,429.088,174.037,23.980,154.166
C02542=1077.437,133.790,429.108,174.036,23.978,154.166
C02543=1077.431,133.541,429.128,174.033,23.975,154.166
C02544=1077.425,133.291,429.149,174.032,23.973,154.166
C02545=1077.419,133.042,429.169,174.030,23.970,154.165
C02546=1077.413,132.793,429.188,174.028,23.968,154.165
C02547=1077.408,132.544,429.209,174.026,23.965,154.165
C02548=1077.402,132.295,429.229,174.025,23.963,154.165
C02549=1077.397,132.046,429.249,174.022,23.961,154.164
C02550=1077.391,131.796,429.269,174.021,23.958,154.164
C02551=1077.385,131.547,429.289,174.019,23.956,154.164
C02552=1077.379,131.299,429.308,174.017,23.954,154.164
C02553=1077.374,131.049,429.328,174.015,23.951,154.163
C02554=1077.368,130.800,429.348,174.014,23.949,154.163
C02555=1077.362,130.551,429.368,174.011,23.946,154.163
C02556=1077.356,130.302,429.387,174.010,23.944,154.163
C02557=1077.351,130.053,429.408,174.008,23.941,154.162
C02558=1077.345,129.803,429.428,174.006,23.940,154.162
C02559=1077.339,129.554,429.448,174.004,23.937,154.162
C02560=1077.333,129.305,429.468,174.003,23.934,154.162
C02561=1077.327,129.056,429.488,174.000,23.932,154.162
C02562=1077.322,128.806,429.507,173.999,23.930,154.161
C02563=1077.316,128.557,429.527,173.997,23.927,154.161
C02564=1077.310,128.308,429.547,173.995,23.925,154.161
C02565=1077.304,128.059,429.567,173.993,23.923,154.161
C02566=1077.298,127.810,429.586,173.992,23.920,154.160
C02567=1077.293,127.529,429.609,173.989,23.918,154.160
C02568=1077.286,127.248,429.631,173.987,23.915,154.160
C02569=1077.280,126.967,429.653,173.986,23.912,154.160
C02570=1077.273,126.686,429.675,173.983,23.910,154.159
C02571=1077.267,126.437,429.695,173.981,23.907,154.159
C02572=1077.262,126.188,429.715,173.980,23.905,154.159
C02573=1077.256,125.938,429.734,173.977,23.902,154.159
C02574=1077.250,125.689,429.754,173.976,23.900,154.158
C02575=1077.245,125.440,429.774,173.975,23.898,154.158
C02576=1077.239,125.191,429.794,173.972,23.895,154.158
C02577=1077.233,124.942,429.813,173.971,23.893,154.158
C02578=1077.228,124.693,429.833,173.969,23.890,154.157
C02579=1077.222,124.443,429.853,173.968,23.888,154.157
C02580=1077.216,124.194,429.873,173.965,23.886,154.157
C02581=1077.210,123.945,429.892,173.964,23.883,154.157
C02582=1077.205,123.696,429.911,173.962,23.881,154.156
C02583=1077.199,123.447,429.931,173.960,23.878,154.156
C02584=1077.193,123.197,429.950,173.958,23.876,154.156
C02585=1077.187,122.948,429.970,173.956,23.874,154.156
C02586=1077.182,122.699,429.990,173.955,23.871,154.155
C02587=1077.176,122.449,430.009,173.953,23.869,154.155
C02588=1077.170,122.200,430.029,173.952,23.866,154.155
C02589=1077.165,121.952,430.048,173.949,23.864,154.155
C02590=1077.159,121.702,430.067,173.948,23.862,154.154
C02591=1077.153,121.453,430.087,173.946,23.859,154.154
C02592=1077.148,121.204,430.107,173.944,23.857,154.154
C02593=1077.142,120.955,430.126,173.942,23.854,154.154
C02594=1077.136,120.706,430.146,173.941,23.852,154.153
C02595=1077.130,120.456,430.165,173.939,23.849,154.153
C02596=1077.125,120.207,430.185,173.937,23.847,154.153
C02597=1077.120,119.959,430.204,173.936,23.845,154.153
C02598=1077.114,119.709,430.224,173.933,23.842,154.152
C02599=1077.109,119.460,430.243,173.932,23.839,154.152
C02600=1077.103,119.211,430.263,173.930,23.837,154.152
C02601=1077.097,118.961,430.282,173.929,23.834,154.151
C02602=1077.091,118.712,430.301,173.927,23.833,154.151
C02603=1077.086,118.463,430.320,173.925,23.830,154.151
C02604=1077.081,118.214,430.340,173.924,23.827,154.151
C02605=1077.075,117.965,430.359,173.921,23.825,154.150
C02606=1077.069,117.716,430.379,173.920,23.822,154.150
C02607=1077.063,117.466,430.398,173.918,23.820,154.150
C02608=1077.057,117.217,430.417,173.916,23.817,154.150
C02609=1077.052,116.968,430.436,173.915,23.815,154.149
C02610=1077.046,116.719,430.456,173.913,23.812,154.149
C02611=1077.041,116.470,430.475,173.911,23.810,154.149
C02612=1077.036,116.220,430.495,173.909,23.807,154.149
C02613=1077.031,115.971,430.514,173.908,23.805,154.148
C02614=1077.025,115.722,430.533,173.906,23.802,154.148
C02615=1077.019,115.472,430.552,173.904,23.800,154.148
C02616=1077.013,115.224,430.572,173.903,23.798,154.147
C02617=1077.008,114.975,430.591,173.901,23.795,154.147
C02618=1077.003,114.725,430.611,173.899,23.793,154.147
C02619=1076.997,114.476,430.630,173.897,23.790,154.147
C02620=1076.991,114.227,430.649,173.896,23.787,154.146
C02621=1076.985,113.977,430.668,173.895,23.785,154.146
C02622=1076.980,113.729,430.687,173.892,23.783,154.146
C02623=1076.974,113.479,430.706,173.891,23.780,154.146
C02624=1076.968,113.230,430.725,173.889,23.778,154.145
C02625=1076.963,112.980,430.744,173.887,23.775,154.145
C02626=1076.957,112.731,430.764,173.886,23.773,154.145
C02627=1076.951,112.483,430.782,173.884,23.770,154.145
C02628=1076.945,112.233,430.801,173.882,23.768,154.144
C02629=1076.940,111.984,430.820,173.880,23.766,154.144
C02630=1076.934,111.734,430.840,173.879,23.763,154.144
C02631=1076.928,111.454,430.861,173.876,23.760,154.144
C02632=1076.921,111.173,430.882,173.875,23.758,154.143
C02633=1076.915,110.891,430.904,173.873,23.755,154.143
C02634=1076.908,110.610,430.925,173.871,23.752,154.143
C02635=1076.902,110.361,430.944,173.869,23.750,154.142
C02636=1076.896,110.112,430.963,173.867,23.747,154.142
C02637=1076.891,109.863,430.982,173.866,23.745,154.142
C02638=1076.885,109.613,431.000,173.864,23.743,154.142
C02639=1076.879,109.364,431.019,173.862,23.740,154.141
C02640=1076.874,109.114,431.039,173.861,23.738,154.141
C02641=1076.869,108.865,431.058,173.859,23.735,154.141
C02642=1076.862,108.616,431.076,173.857,23.733,154.141
C02643=1076.856,108.367,431.095,173.856,23.730,154.140
C02644=1076.851,108.117,431.115,173.854,23.728,154.140
C02645=1076.845,107.869,431.133,173.852,23.726,154.140
C02646=1076.839,107.619,431.151,173.851,23.723,154.140
C02647=1076.834,107.370,431.171,173.849,23.720,154.139
C02648=1076.828,107.121,431.189,173.847,23.718,154.139
C02649=1076.822,106.872,431.208,173.845,23.715,154.139
C02650=1076.816,106.623,431.227,173.844,23.713,154.138
C02651=1076.811,106.374,431.246,173.843,23.711,154.138
C02652=1076.805,106.124,431.264,173.840,23.708,154.138
C02653=1076.799,105.875,431.283,173.839,23.706,154.138
C02654=1076.794,105.626,431.302,173.838,23.704,154.137
C02655=1076.788,105.377,431.321,173.835,23.701,154.137
C02656=1076.782,105.127,431.339,173.834,23.698,154.137
C02657=1076.777,104.878,431.358,173.832,23.696,154.137
C02658=1076.771,104.629,431.377,173.831,23.693,154.136
C02659=1076.765,104.380,431.396,173.829,23.691,154.136
C02660=1076.760,104.130,431.414,173.827,23.688,154.136
C02661=1076.754,103.881,431.433,173.826,23.686,154.135
C02662=1076.748,103.632,431.452,173.824,23.683,154.135
C02663=1076.743,103.383,431.471,173.822,23.681,154.135
C02664=1076.737,103.133,431.489,173.821,23.678,154.135
C02665=1076.731,102.884,431.508,173.820,23.676,154.134
C02666=1076.725,102.635,431.526,173.817,23.673,154.134
C02667=1076.720,102.385,431.545,173.816,23.671,154.134
C02668=1076.715,102.137,431.564,173.814,23.669,154.134
C02669=1076.708,101.887,431.582,173.812,23.666,154.133
C02670=1076.703,101.637,431.601,173.811,23.664,154.133
C02671=1076.697,101.389,431.619,173.809,23.661,154.133
C02672=1076.692,101.139,431.638,173.807,23.659,154.133
C02673=1076.686,100.890,431.656,173.806,23.656,154.132
C02674=1076.680,100.641,431.675,173.804,23.654,154.132
C02675=1076.674,100.391,431.693,173.803,23.651,154.132
C02676=1076.669,100.143,431.712,173.801,23.649,154.131
C02677=1076.663,99.893,431.730,173.799,23.646,154.131
C02678=1076.657,99.644,431.748,173.798,23.644,154.131
C02679=1076.651,99.395,431.767,173.796,23.641,154.131
C02680=1076.645,99.145,431.785,173.794,23.639,154.130
C02681=1076.640,98.896,431.804,173.793,23.637,154.130
C02682=1076.634,98.647,431.822,173.791,23.634,154.130
C02683=1076.628,98.398,431.841,173.789,23.631,154.130
C02684=1076.623,98.148,431.859,173.788,23.629,154.129
C02685=1076.616,97.899,431.878,173.787,23.627,154.129
C02686=1076.611,97.650,431.895,173.784,23.624,154.129
C02687=1076.605,97.401,431.914,173.783,23.622,154.128
C02688=1076.599,97.151,431.932,173.781,23.619,154.128
C02689=1076.594,96.902,431.951,173.780,23.616,154.128
C02690=1076.588,96.652,431.969,173.778,23.614,154.128
C02691=1076.582,96.404,431.987,173.776,23.611,154.127
C02692=1076.577,96.154,432.006,173.775,23.609,154.127
C02693=1076.571,95.905,432.023,173.773,23.607,154.127
C02694=1076.565,95.656,432.042,173.771,23.604,154.126
C02695=1076.559,95.375,432.063,173.770,23.601,154.126
C02696=1076.552,95.093,432.083,173.768,23.599,154.126
C02697=1076.546,94.813,432.104,173.766,23.596,154.126
C02698=1076.539,94.531,432.124,173.764,23.593,154.125
C02699=1076.534,94.282,432.142,173.763,23.591,154.125
C02700=1076.528,94.033,432.161,173.761,23.588,154.125
C02701=1076.522,93.784,432.179,173.759,23.585,154.124
C02702=1076.517,93.534,432.198,173.758,23.583,154.124
C02703=1076.511,93.285,432.215,173.756,23.580,154.124
C02704=1076.505,93.035,432.233,173.755,23.578,154.124
C02705=1076.500,92.787,432.252,173.753,23.575,154.123
C02706=1076.494,92.537,432.270,173.751,23.573,154.123
C02707=1076.488,92.288,432.288,173.750,23.570,154.123
C02708=1076.482,92.039,432.306,173.748,23.568,154.122
C02709=1076.477,91.789,432.325,173.746,23.565,154.122
C02710=1076.471,91.540,432.343,173.745,23.563,154.122
C02711=1076.465,91.291,432.360,173.744,23.560,154.122
C02712=1076.460,91.041,432.379,173.741,23.558,154.121
C02713=1076.454,90.792,432.397,173.740,23.555,154.121
C02714=1076.448,90.542,432.415,173.739,23.553,154.121
C02715=1076.443,90.293,432.432,173.737,23.550,154.121
C02716=1076.436,90.044,432.451,173.735,23.548,154.120
C02717=1076.431,89.795,432.469,173.734,23.545,154.120
C02718=1076.425,89.546,432.487,173.733,23.543,154.120
C02719=1076.419,89.296,432.504,173.731,23.540,154.119
C02720=1076.414,89.046,432.523,173.729,23.538,154.119
C02721=1076.408,88.798,432.541,173.728,23.535,154.119
C02722=1076.402,88.548,432.559,173.726,23.533,154.119
C02723=1076.396,88.299,432.576,173.724,23.530,154.118
C02724=1076.390,88.049,432.594,173.723,23.528,154.118
C02725=1076.385,87.800,432.612,173.721,23.526,154.118
C02726=1076.378,87.551,432.630,173.719,23.523,154.118
C02727=1076.373,87.302,432.648,173.718,23.521,154.117
C02728=1076.367,87.053,432.666,173.716,23.518,154.117
C02729=1076.361,86.803,432.684,173.715,23.516,154.117
C02730=1076.355,86.554,432.701,173.713,23.513,154.116
C02731=1076.349,86.305,432.719,173.712,23.511,154.116
C02732=1076.344,86.056,432.737,173.710,23.508,154.116
C02733=1076.338,85.806,432.755,173.708,23.506,154.116
C02734=1076.333,85.557,432.773,173.707,23.503,154.115
C02735=1076.327,85.308,432.790,173.705,23.501,154.115
C02736=1076.321,85.058,432.808,173.704,23.498,154.115
C02737=1076.315,84.809,432.827,173.702,23.496,154.114
C02738=1076.309,84.560,432.845,173.700,23.493,154.114
C02739=1076.304,84.311,432.862,173.699,23.491,154.114
C02740=1076.298,84.062,432.880,173.698,23.488,154.114
C02741=1076.292,83.812,432.898,173.696,23.486,154.113
C02742=1076.287,83.563,432.915,173.694,23.483,154.113
C02743=1076.281,83.313,432.933,173.693,23.480,154.113
C02744=1076.275,83.064,432.951,173.692,23.478,154.112
C02745=1076.270,82.815,432.968,173.689,23.475,154.112
C02746=1076.263,82.565,432.986,173.688,23.473,154.112
C02747=1076.258,82.316,433.004,173.687,23.470,154.112
C02748=1076.252,82.067,433.021,173.686,23.468,154.111
C02749=1076.246,81.817,433.039,173.683,23.465,154.111
C02750=1076.241,81.568,433.057,173.682,23.463,154.111
C02751=1076.235,81.319,433.074,173.681,23.460,154.110
C02752=1076.229,81.069,433.092,173.678,23.457,154.110
C02753=1076.224,80.820,433.109,173.677,23.455,154.110
C02754=1076.218,80.571,433.127,173.676,23.453,154.110
C02755=1076.212,80.321,433.145,173.675,23.450,154.109
C02756=1076.207,80.072,433.162,173.672,23.448,154.109
C02757=1076.201,79.823,433.180,173.671,23.445,154.109
C02758=1076.195,79.573,433.198,173.670,23.442,154.108
C02759=1076.189,79.292,433.218,173.668,23.439,154.108
C02760=1076.182,79.011,433.236,173.666,23.437,154.108
C02761=1076.176,78.730,433.257,173.664,23.434,154.107
C02762=1076.170,78.449,433.277,173.662,23.431,154.107
C02763=1076.164,78.200,433.294,173.661,23.429,154.107
C02764=1076.158,77.950,433.311,173.660,23.426,154.107
C02765=1076.152,77.701,433.328,173.659,23.423,154.106
C02766=1076.146,77.452,433.346,173.656,23.420,154.106
C02767=1076.140,77.203,433.364,173.655,23.418,154.106
C02768=1076.135,76.953,433.381,173.654,23.416,154.105
C02769=1076.128,76.703,433.398,173.652,23.413,154.105
C02770=1076.123,76.454,433.416,173.650,23.410,154.105
C02771=1076.117,76.205,433.433,173.649,23.408,154.104
C02772=1076.112,75.956,433.451,173.648,23.406,154.104
C02773=1076.106,75.706,433.468,173.645,23.403,154.104
C02774=1076.100,75.457,433.485,173.644,23.400,154.104
C02775=1076.094,75.208,433.502,173.643,23.398,154.103
C02776=1076.088,74.958,433.520,173.642,23.396,154.103
C02777=1076.083,74.709,433.537,173.639,23.393,154.103
C02778=1076.077,74.460,433.554,173.638,23.391,154.102
C02779=1076.071,74.211,433.572,173.637,23.388,154.102
C02780=1076.065,73.961,433.589,173.635,23.386,154.102
C02781=1076.060,73.712,433.607,173.633,23.383,154.102
C02782=1076.054,73.463,433.624,173.632,23.381,154.101
C02783=1076.048,73.214,433.641,173.631,23.378,154.101
C02784=1076.042,72.963,433.658,173.629,23.375,154.101
C02785=1076.037,72.714,433.676,173.627,23.373,154.100
C02786=1076.031,72.465,433.692,173.626,23.370,154.100
C02787=1076.025,72.216,433.710,173.625,23.368,154.100
C02788=1076.019,71.966,433.728,173.623,23.365,154.100
C02789=1076.013,71.717,433.744,173.621,23.362,154.099
C02790=1076.008,71.468,433.761,173.620,23.360,154.099
C02791=1076.002,71.219,433.779,173.619,23.358,154.099
C02792=1075.996,70.970,433.795,173.617,23.355,154.098
C02793=1075.990,70.720,433.813,173.615,23.352,154.098
C02794=1075.985,70.470,433.830,173.614,23.350,154.098
C02795=1075.979,70.221,433.848,173.613,23.348,154.098
C02796=1075.973,69.972,433.864,173.610,23.345,154.097
C02797=1075.968,69.723,433.881,173.609,23.342,154.097
C02798=1075.961,69.473,433.899,173.608,23.340,154.097
C02799=1075.956,69.224,433.916,173.607,23.337,154.096
C02800=1075.950,68.975,433.933,173.605,23.334,154.096
C02801=1075.944,68.725,433.949,173.603,23.332,154.096
C02802=1075.939,68.476,433.967,173.602,23.330,154.095
C02803=1075.932,68.226,433.984,173.601,23.327,154.095
C02804=1075.927,67.977,434.001,173.599,23.324,154.095
C02805=1075.921,67.728,434.017,173.597,23.322,154.095
C02806=1075.915,67.479,434.035,173.596,23.320,154.094
C02807=1075.910,67.229,434.052,173.595,23.317,154.094
C02808=1075.904,66.979,434.069,173.592,23.314,154.094
C02809=1075.898,66.730,434.086,173.591,23.312,154.093
C02810=1075.892,66.481,434.102,173.590,23.310,154.093
C02811=1075.887,66.232,434.120,173.589,23.307,154.093
C02812=1075.881,65.982,434.136,173.587,23.304,154.093
C02813=1075.875,65.733,434.154,173.585,23.301,154.092
C02814=1075.868,65.483,434.170,173.584,23.299,154.092
C02815=1075.863,65.233,434.187,173.583,23.297,154.092
C02816=1075.857,64.985,434.204,173.581,23.294,154.091
C02817=1075.852,64.735,434.221,173.579,23.291,154.091
C02818=1075.846,64.486,434.238,173.578,23.289,154.091
C02819=1075.840,64.237,434.255,173.577,23.287,154.091
C02820=1075.834,63.987,434.271,173.574,23.284,154.090
C02821=1075.828,63.738,434.288,173.573,23.281,154.090
C02822=1075.822,63.488,434.305,173.572,23.279,154.090
C02823=1075.816,63.207,434.324,173.570,23.276,154.089
C02824=1075.809,62.926,434.343,173.569,23.273,154.089
C02825=1075.802,62.645,434.361,173.566,23.271,154.089
C02826=1075.795,62.364,434.381,173.565,23.268,154.088
C02827=1075.789,62.115,434.397,173.564,23.265,154.088
C02828=1075.783,61.865,434.413,173.562,23.262,154.088
C02829=1075.778,61.615,434.431,173.561,23.260,154.088
C02830=1075.771,61.366,434.448,173.559,23.258,154.087
C02831=1075.765,61.117,434.464,173.558,23.255,154.087
C02832=1075.760,60.867,434.481,173.557,23.253,154.087
C02833=1075.754,60.618,434.497,173.554,23.250,154.086
C02834=1075.748,60.369,434.514,173.553,23.248,154.086
C02835=1075.742,60.120,434.530,173.552,23.245,154.086
C02836=1075.737,59.870,434.547,173.551,23.243,154.086
C02837=1075.730,59.620,434.564,173.548,23.240,154.085
C02838=1075.724,59.371,434.581,173.547,23.238,154.085
C02839=1075.719,59.122,434.598,173.546,23.235,154.085
C02840=1075.713,58.872,434.614,173.545,23.233,154.084
C02841=1075.707,58.623,434.630,173.542,23.230,154.084
C02842=1075.701,58.374,434.646,173.541,23.228,154.084
C02843=1075.695,58.125,434.664,173.540,23.225,154.084
C02844=1075.690,57.875,434.680,173.539,23.223,154.083
C02845=1075.684,57.626,434.696,173.537,23.220,154.083
C02846=1075.678,57.377,434.713,173.535,23.217,154.083
C02847=1075.672,57.127,434.729,173.534,23.215,154.082
C02848=1075.666,56.878,434.746,173.533,23.212,154.082
C02849=1075.660,56.628,434.762,173.531,23.210,154.082
C02850=1075.654,56.379,434.779,173.529,23.207,154.081
C02851=1075.648,56.129,434.796,173.528,23.205,154.081
C02852=1075.642,55.880,434.812,173.527,23.202,154.081
C02853=1075.637,55.631,434.829,173.525,23.200,154.081
C02854=1075.631,55.381,434.845,173.524,23.197,154.080
C02855=1075.625,55.132,434.861,173.522,23.194,154.080
C02856=1075.619,54.882,434.878,173.521,23.192,154.080
C02857=1075.613,54.633,434.894,173.519,23.190,154.079
C02858=1075.608,54.383,434.911,173.518,23.187,154.079
C02859=1075.602,54.134,434.927,173.516,23.184,154.079
C02860=1075.596,53.885,434.943,173.515,23.182,154.079
C02861=1075.590,53.635,434.960,173.514,23.179,154.078
C02862=1075.584,53.386,434.976,173.512,23.177,154.078
C02863=1075.578,53.136,434.992,173.511,23.174,154.078
C02864=1075.573,52.887,435.009,173.509,23.171,154.077
C02865=1075.567,52.638,435.025,173.508,23.169,154.077
C02866=1075.561,52.388,435.042,173.506,23.167,154.077
C02867=1075.555,52.139,435.058,173.505,23.164,154.077
C02868=1075.549,51.889,435.074,173.504,23.161,154.076
C02869=1075.544,51.640,435.091,173.502,23.158,154.076
C02870=1075.538,51.391,435.107,173.500,23.156,154.076
C02871=1075.532,51.141,435.123,173.499,23.154,154.075
C02872=1075.527,50.892,435.140,173.498,23.151,154.075
C02873=1075.521,50.643,435.156,173.496,23.148,154.075
C02874=1075.515,50.394,435.172,173.494,23.146,154.074
C02875=1075.509,50.144,435.188,173.493,23.144,154.074
C02876=1075.503,49.895,435.205,173.492,23.141,154.074
C02877=1075.497,49.646,435.221,173.491,23.138,154.073
C02878=1075.492,49.395,435.237,173.489,23.135,154.073
C02879=1075.486,49.146,435.253,173.487,23.133,154.073
C02880=1075.480,48.897,435.269,173.486,23.131,154.073
C02881=1075.474,48.647,435.286,173.485,23.128,154.072
C02882=1075.469,48.398,435.302,173.484,23.125,154.072
C02883=1075.463,48.149,435.318,173.481,23.122,154.072
C02884=1075.457,47.900,435.334,173.480,23.120,154.071
C02885=1075.452,47.650,435.350,173.479,23.118,154.071
C02886=1075.446,47.400,435.367,173.478,23.115,154.071
C02887=1075.440,47.119,435.385,173.476,23.112,154.070
C02888=1075.433,46.837,435.403,173.474,23.109,154.070
C02889=1075.426,46.556,435.421,173.472,23.106,154.070
C02890=1075.420,46.275,435.439,173.471,23.103,154.069
C02891=1075.414,46.026,435.455,173.470,23.101,154.069
C02892=1075.409,45.776,435.471,173.468,23.098,154.069
C02893=1075.403,45.526,435.488,173.467,23.096,154.068
C02894=1075.397,45.277,435.504,173.465,23.093,154.068
C02895=1075.392,45.028,435.520,173.464,23.090,154.068
C02896=1075.386,44.778,435.536,173.463,23.088,154.067
C02897=1075.381,44.529,435.552,173.461,23.085,154.067
C02898=1075.375,44.280,435.568,173.459,23.082,154.067
C02899=1075.369,44.030,435.584,173.458,23.080,154.067
C02900=1075.363,43.780,435.600,173.457,23.077,154.066
C02901=1075.357,43.531,435.616,173.456,23.075,154.066
C02902=1075.351,43.282,435.632,173.454,23.072,154.066
C02903=1075.345,43.032,435.648,173.452,23.069,154.065
C02904=1075.340,42.783,435.664,173.451,23.067,154.065
C02905=1075.334,42.534,435.680,173.450,23.065,154.065
C02906=1075.328,42.284,435.695,173.449,23.062,154.065
C02907=1075.323,42.034,435.712,173.446,23.059,154.064
C02908=1075.317,41.785,435.728,173.445,23.057,154.064
C02909=1075.310,41.535,435.743,173.444,23.055,154.064
C02910=1075.305,41.287,435.759,173.443,23.052,154.063
C02911=1075.299,41.037,435.775,173.442,23.049,154.063
C02912=1075.293,40.787,435.791,173.440,23.047,154.063
C02913=1075.287,40.538,435.807,173.438,23.044,154.062
C02914=1075.282,40.288,435.822,173.437,23.042,154.062
C02915=1075.276,40.039,435.839,173.436,23.039,154.062
C02916=1075.270,39.790,435.855,173.434,23.037,154.062
C02917=1075.264,39.540,435.869,173.433,23.034,154.061
C02918=1075.258,39.291,435.886,173.431,23.031,154.061
C02919=1075.252,39.041,435.901,173.430,23.029,154.061
C02920=1075.247,38.792,435.917,173.428,23.026,154.060
C02921=1075.241,38.542,435.933,173.427,23.024,154.060
C02922=1075.235,38.293,435.949,173.426,23.021,154.060
C02923=1075.230,38.043,435.965,173.424,23.018,154.060
C02924=1075.223,37.794,435.980,173.423,23.016,154.059
C02925=1075.218,37.545,435.995,173.421,23.014,154.059
C02926=1075.212,37.296,436.012,173.420,23.011,154.059
C02927=1075.206,37.046,436.027,173.419,23.009,154.058
C02928=1075.200,36.797,436.043,173.418,23.006,154.058
C02929=1075.194,36.547,436.058,173.415,23.003,154.058
C02930=1075.189,36.298,436.074,173.414,23.001,154.057
C02931=1075.182,36.048,436.089,173.413,22.998,154.057
C02932=1075.176,35.799,436.105,173.412,22.996,154.057
C02933=1075.171,35.549,436.121,173.410,22.993,154.057
C02934=1075.164,35.300,436.137,173.408,22.990,154.056
C02935=1075.159,35.051,436.152,173.407,22.988,154.056
C02936=1075.153,34.801,436.168,173.406,22.986,154.056
C02937=1075.147,34.552,436.183,173.404,22.983,154.055
C02938=1075.141,34.302,436.199,173.403,22.981,154.055
C02939=1075.136,34.053,436.214,173.402,22.978,154.055
C02940=1075.129,33.803,436.229,173.400,22.976,154.055
C02941=1075.123,33.554,436.246,173.398,22.973,154.054
C02942=1075.118,33.304,436.261,173.397,22.970,154.054
C02943=1075.112,33.055,436.276,173.396,22.968,154.054
C02944=1075.106,32.806,436.292,173.395,22.965,154.053
C02945=1075.100,32.556,436.308,173.393,22.962,154.053
C02946=1075.094,32.306,436.323,173.391,22.960,154.053
C02947=1075.089,32.057,436.338,173.390,22.958,154.052
C02948=1075.083,31.807,436.354,173.389,22.955,154.052
C02949=1075.077,31.558,436.369,173.388,22.953,154.052
C02950=1075.071,31.309,436.385,173.386,22.950,154.052
C02951=1075.064,31.028,436.402,173.384,22.947,154.051
C02952=1075.058,30.745,436.419,173.383,22.945,154.051
C02953=1075.052,30.464,436.437,173.381,22.941,154.051
C02954=1075.045,30.183,436.454,173.380,22.939,154.050
C02955=1075.039,29.933,436.469,173.379,22.936,154.050
C02956=1075.033,29.685,436.485,173.376,22.934,154.050
C02957=1075.027,29.435,436.500,173.375,22.931,154.049
C02958=1075.021,29.185,436.516,173.374,22.928,154.049
C02959=1075.016,28.936,436.530,173.373,22.926,154.049
C02960=1075.010,28.686,436.547,173.372,22.923,154.048
C02961=1075.003,28.437,436.562,173.370,22.921,154.048
C02962=1074.998,28.187,436.577,173.368,22.918,154.048
C02963=1074.992,27.938,436.592,173.367,22.916,154.048
C02964=1074.986,27.688,436.607,173.366,22.913,154.047
C02965=1074.980,27.439,436.623,173.364,22.911,154.047
C02966=1074.975,27.190,436.638,173.363,22.908,154.047
C02967=1074.968,26.940,436.653,173.362,22.906,154.046
C02968=1074.963,26.691,436.668,173.360,22.903,154.046
C02969=1074.957,26.441,436.683,173.358,22.901,154.046
C02970=1074.951,26.192,436.699,173.357,22.898,154.046
C02971=1074.945,25.943,436.714,173.356,22.896,154.045
C02972=1074.939,25.693,436.729,173.355,22.893,154.045
C02973=1074.933,25.443,436.745,173.353,22.891,154.045
C02974=1074.927,25.194,436.759,173.351,22.888,154.045
C02975=1074.922,24.944,436.775,173.350,22.886,154.044
C02976=1074.915,24.694,436.790,173.349,22.883,154.044
C02977=1074.910,24.445,436.805,173.348,22.880,154.044
C02978=1074.904,24.195,436.820,173.346,22.878,154.043
C02979=1074.897,23.946,436.835,173.345,22.875,154.043
C02980=1074.892,23.697,436.851,173.343,22.873,154.043
C02981=1074.886,23.448,436.866,173.342,22.870,154.042
C02982=1074.881,23.198,436.881,173.341,22.868,154.042
C02983=1074.874,22.949,436.896,173.339,22.865,154.042
C02984=1074.868,22.699,436.911,173.338,22.863,154.042
C02985=1074.863,22.450,436.926,173.337,22.860,154.041
C02986=1074.856,22.200,436.941,173.335,22.858,154.041
C02987=1074.851,21.951,436.956,173.333,22.855,154.041
C02988=1074.845,21.701,436.971,173.332,22.853,154.040
C02989=1074.839,21.451,436.986,173.331,22.850,154.040
C02990=1074.834,21.202,437.001,173.330,22.848,154.040
C02991=1074.827,20.953,437.016,173.328,22.845,154.040
C02992=1074.821,20.704,437.030,173.326,22.843,154.039
C02993=1074.816,20.454,437.046,173.325,22.840,154.039
C02994=1074.810,20.205,437.061,173.324,22.838,154.039
C02995=1074.804,19.955,437.076,173.322,22.835,154.038
C02996=1074.798,19.705,437.091,173.321,22.833,154.038
C02997=1074.792,19.456,437.106,173.320,22.830,154.038
C02998=1074.786,19.206,437.121,173.319,22.828,154.038
C02999=1074.781,18.957,437.135,173.316,22.825,154.037
C03000=1074.775,18.707,437.150,173.315,22.823,154.037
C03001=1074.769,18.458,437.165,173.314,22.820,154.037
C03002=1074.762,18.208,437.180,173.313,22.818,154.037
C03003=1074.757,17.958,437.195,173.311,22.815,154.036
C03004=1074.751,17.709,437.210,173.310,22.813,154.036
C03005=1074.745,17.460,437.225,173.308,22.810,154.036
C03006=1074.739,17.211,437.239,173.307,22.808,154.035
C03007=1074.733,16.961,437.255,173.306,22.805,154.035
C03008=1074.728,16.711,437.269,173.305,22.802,154.035
C03009=1074.721,16.462,437.284,173.303,22.800,154.034
C03010=1074.716,16.213,437.298,173.302,22.798,154.034
C03011=1074.710,15.963,437.314,173.300,22.795,154.034
C03012=1074.704,15.714,437.328,173.299,22.792,154.034
C03013=1074.698,15.464,437.343,173.297,22.790,154.033
C03014=1074.692,15.214,437.357,173.296,22.787,154.033
C03015=1074.686,14.934,437.375,173.295,22.785,154.033
C03016=1074.679,14.654,437.391,173.293,22.782,154.032
C03017=1074.672,14.375,437.407,173.292,22.779,154.032
C03018=1074.666,14.094,437.424,173.289,22.776,154.032
C03019=1074.660,13.845,437.439,173.288,22.774,154.032
C03020=1074.654,13.595,437.453,173.287,22.771,154.031
C03021=1074.648,13.346,437.467,173.286,22.769,154.031
C03022=1074.642,13.096,437.482,173.284,22.767,154.031
C03023=1074.636,12.847,437.497,173.283,22.764,154.030
C03024=1074.630,12.597,437.511,173.281,22.761,154.030
C03025=1074.624,12.348,437.526,173.280,22.759,154.030
C03026=1074.618,12.098,437.541,173.278,22.757,154.030
C03027=1074.612,11.849,437.555,173.277,22.755,154.029
C03028=1074.606,11.599,437.570,173.276,22.752,154.029
C03029=1074.600,11.350,437.584,173.275,22.750,154.029
C03030=1074.594,11.100,437.599,173.273,22.747,154.029
C03031=1074.588,10.851,437.613,173.271,22.744,154.028
C03032=1074.582,10.601,437.628,173.270,22.742,154.028
C03033=1074.576,10.352,437.642,173.269,22.739,154.028
C03034=1074.570,10.102,437.657,173.268,22.737,154.027
C03035=1074.564,9.853,437.671,173.266,22.735,154.027
C03036=1074.558,9.603,437.686,173.265,22.732,154.027
C03037=1074.552,9.354,437.700,173.264,22.730,154.027
C03038=1074.546,9.104,437.715,173.261,22.727,154.026
C03039=1074.540,8.854,437.729,173.260,22.725,154.026
C03040=1074.534,8.605,437.744,173.259,22.723,154.026
C03041=1074.528,8.356,437.758,173.258,22.720,154.026
C03042=1074.522,8.106,437.773,173.256,22.718,154.025
C03043=1074.516,7.857,437.787,173.255,22.715,154.025
C03044=1074.511,7.607,437.801,173.254,22.713,154.025
C03045=1074.505,7.357,437.816,173.252,22.710,154.024
C03046=1074.499,7.108,437.830,173.251,22.708,154.024
C03047=1074.493,6.858,437.845,173.249,22.705,154.024
C03048=1074.487,6.609,437.859,173.248,22.703,154.024
C03049=1074.481,6.359,437.874,173.247,22.700,154.023
C03050=1074.475,6.110,437.888,173.246,22.698,154.023
C03051=1074.470,5.860,437.902,173.244,22.696,154.023
C03052=1074.463,5.611,437.917,173.242,22.693,154.023
C03053=1074.457,5.362,437.930,173.241,22.691,154.022
C03054=1074.451,5.112,437.945,173.240,22.688,154.022
C03055=1074.445,4.862,437.959,173.238,22.686,154.022
C03056=1074.439,4.613,437.974,173.237,22.683,154.021
C03057=1074.433,4.363,437.988,173.236,22.681,154.021
C03058=1074.428,4.114,438.002,173.235,22.678,154.021
C03059=1074.422,3.865,438.016,173.232,22.676,154.021
C03060=1074.416,3.614,438.031,173.231,22.673,154.020
C03061=1074.410,3.365,438.045,173.230,22.671,154.020
C03062=1074.404,3.115,438.059,173.229,22.668,154.020
C03063=1074.398,2.866,438.074,173.228,22.666,154.020
C03064=1074.393,2.616,438.088,173.226,22.663,154.019
C03065=1074.386,2.367,438.103,173.225,22.661,154.019
C03066=1074.381,2.117,438.117,173.223,22.659,154.019
C03067=1074.375,1.868,438.130,173.221,22.656,154.019
C03068=1074.368,1.618,438.145,173.220,22.654,154.018
C03069=1074.363,1.369,438.159,173.219,22.651,154.018
C03070=1074.357,1.120,438.173,173.218,22.649,154.018
C03071=1074.352,0.870,438.187,173.216,22.646,154.017
C03072=1074.346,0.620,438.201,173.215,22.644,154.017
C03073=1074.340,0.371,438.216,173.213,22.641,154.017
C03074=1074.334,0.121,438.230,173.212,22.639,154.017
C03075=1074.328,-0.129,438.244,173.211,22.636,154.016
C03076=1074.322,-0.378,438.259,173.209,22.634,154.016
C03077=1074.316,-0.627,438.272,173.208,22.631,154.016
C03078=1074.311,-0.877,438.286,173.207,22.629,154.016
C03079=1074.304,-1.155,438.302,173.205,22.626,154.015
C03080=1074.297,-1.433,438.318,173.204,22.624,154.015
C03081=1074.291,-1.711,438.334,173.202,22.621,154.015
C03082=1074.285,-1.990,438.349,173.200,22.618,154.014
C03083=1074.278,-2.238,438.363,173.199,22.616,154.014
C03084=1074.273,-2.488,438.377,173.198,22.613,154.014
C03085=1074.267,-2.737,438.391,173.196,22.611,154.014
C03086=1074.261,-2.988,438.405,173.195,22.609,154.013
C03087=1074.255,-3.237,438.420,173.193,22.606,154.013
C03088=1074.250,-3.486,438.434,173.192,22.603,154.013
C03089=1074.243,-3.736,438.447,173.191,22.601,154.012
C03090=1074.238,-3.986,438.461,173.189,22.598,154.012
C03091=1074.232,-4.235,438.474,173.188,22.596,154.012
C03092=1074.226,-4.484,438.489,173.187,22.594,154.012
C03093=1074.220,-4.734,438.503,173.185,22.592,154.011
C03094=1074.213,-4.984,438.516,173.184,22.589,154.011
C03095=1074.208,-5.233,438.530,173.182,22.587,154.011
C03096=1074.202,-5.483,438.545,173.181,22.584,154.011
C03097=1074.195,-5.732,438.559,173.179,22.582,154.010
C03098=1074.190,-5.982,438.572,173.178,22.579,154.010
C03099=1074.184,-6.231,438.586,173.177,22.577,154.010
C03100=1074.178,-6.481,438.600,173.176,22.575,154.010
C03101=1074.172,-6.731,438.614,173.174,22.573,154.009
C03102=1074.166,-6.980,438.627,173.172,22.570,154.009
C03103=1074.160,-7.230,438.641,173.171,22.567,154.009
C03104=1074.154,-7.480,438.655,173.170,22.565,154.009
C03105=1074.148,-7.729,438.669,173.168,22.563,154.008
C03106=1074.142,-7.978,438.682,173.167,22.561,154.008
C03107=1074.136,-8.227,438.696,173.166,22.558,154.008
C03108=1074.130,-8.478,438.711,173.164,22.556,154.008
C03109=1074.124,-8.727,438.724,173.163,22.554,154.007
C03110=1074.118,-8.976,438.738,173.161,22.551,154.007
C03111=1074.112,-9.226,438.751,173.160,22.548,154.007
C03112=1074.106,-9.476,438.765,173.159,22.546,154.007
C03113=1074.101,-9.726,438.779,173.157,22.544,154.006
C03114=1074.094,-9.975,438.792,173.156,22.542,154.006
C03115=1074.089,-10.224,438.806,173.155,22.539,154.006
C03116=1074.083,-10.474,438.819,173.153,22.537,154.006
C03117=1074.077,-10.724,438.834,173.152,22.535,154.005
C03118=1074.070,-10.973,438.847,173.150,22.532,154.005
C03119=1074.065,-11.223,438.861,173.149,22.530,154.005
C03120=1074.059,-11.472,438.874,173.147,22.527,154.005
C03121=1074.053,-11.722,438.888,173.146,22.525,154.004
C03122=1074.047,-11.971,438.901,173.145,22.523,154.004
C03123=1074.041,-12.221,438.915,173.144,22.520,154.004
C03124=1074.035,-12.471,438.929,173.142,22.518,154.004
C03125=1074.029,-12.720,438.943,173.140,22.515,154.003
C03126=1074.024,-12.970,438.956,173.139,22.513,154.003
C03127=1074.018,-13.219,438.970,173.138,22.511,154.003
C03128=1074.012,-13.468,438.984,173.136,22.508,154.003
C03129=1074.006,-13.718,438.997,173.135,22.506,154.002
C03130=1074.000,-13.968,439.011,173.134,22.504,154.002
C03131=1073.994,-14.217,439.024,173.132,22.501,154.002
C03132=1073.988,-14.467,439.038,173.131,22.499,154.002
C03133=1073.982,-14.717,439.051,173.129,22.496,154.001
C03134=1073.977,-14.966,439.065,173.128,22.494,154.001
C03135=1073.971,-15.216,439.078,173.126,22.492,154.001
C03136=1073.964,-15.465,439.091,173.125,22.489,154.001
C03137=1073.959,-15.714,439.105,173.124,22.487,154.000
C03138=1073.952,-15.964,439.119,173.123,22.485,154.000
C03139=1073.946,-16.214,439.132,173.121,22.482,154.000
C03140=1073.941,-16.464,439.145,173.120,22.481,154.000
C03141=1073.934,-16.713,439.158,173.118,22.478,154.000
C03142=1073.928,-16.962,439.172,173.116,22.476,153.999
C03143=1073.922,-17.239,439.187,173.115,22.473,153.999
C03144=1073.915,-17.516,439.202,173.114,22.471,153.999
C03145=1073.908,-17.792,439.217,173.112,22.468,153.999
C03146=1073.902,-18.068,439.231,173.111,22.466,153.998
C03147=1073.895,-18.317,439.245,173.109,22.463,153.998
C03148=1073.890,-18.568,439.258,173.108,22.461,153.998
C03149=1073.884,-18.817,439.271,173.107,22.459,153.998
C03150=1073.878,-19.066,439.284,173.105,22.456,153.997
C03151=1073.872,-19.316,439.298,173.103,22.454,153.997
C03152=1073.866,-19.566,439.311,173.102,22.451,153.997
C03153=1073.860,-19.816,439.324,173.101,22.449,153.997
C03154=1073.853,-20.065,439.338,173.099,22.447,153.996
C03155=1073.848,-20.314,439.351,173.098,22.445,153.996
C03156=1073.842,-20.564,439.364,173.097,22.443,153.996
C03157=1073.836,-20.814,439.377,173.096,22.440,153.996
C03158=1073.830,-21.063,439.391,173.093,22.437,153.995
C03159=1073.824,-21.313,439.404,173.092,22.436,153.995
C03160=1073.818,-21.562,439.417,173.091,22.433,153.995
C03161=1073.812,-21.812,439.430,173.089,22.431,153.995
C03162=1073.807,-22.062,439.443,173.088,22.429,153.995
C03163=1073.801,-22.311,439.457,173.087,22.426,153.994
C03164=1073.794,-22.560,439.470,173.085,22.424,153.994
C03165=1073.788,-22.810,439.482,173.084,22.422,153.994
C03166=1073.783,-23.060,439.496,173.083,22.420,153.994
C03167=1073.777,-23.309,439.510,173.081,22.417,153.993
C03168=1073.771,-23.559,439.522,173.079,22.415,153.993
C03169=1073.765,-23.808,439.535,173.078,22.413,153.993
C03170=1073.759,-24.058,439.549,173.077,22.410,153.993
C03171=1073.753,-24.308,439.562,173.075,22.408,153.993
C03172=1073.747,-24.557,439.575,173.074,22.406,153.992
C03173=1073.741,-24.807,439.588,173.073,22.403,153.992
C03174=1073.736,-25.056,439.602,173.072,22.402,153.992
C03175=1073.729,-25.306,439.615,173.069,22.399,153.992
C03176=1073.723,-25.556,439.627,173.068,22.397,153.991
C03177=1073.717,-25.805,439.641,173.067,22.394,153.991
C03178=1073.711,-26.055,439.653,173.066,22.392,153.991
C03179=1073.706,-26.304,439.667,173.064,22.390,153.991
C03180=1073.700,-26.554,439.680,173.063,22.387,153.990
C03181=1073.694,-26.803,439.693,173.062,22.386,153.990
C03182=1073.688,-27.053,439.705,173.060,22.383,153.990
C03183=1073.682,-27.303,439.719,173.059,22.381,153.990
C03184=1073.676,-27.552,439.731,173.057,22.378,153.990
C03185=1073.670,-27.802,439.745,173.055,22.376,153.989
C03186=1073.664,-28.052,439.757,173.054,22.374,153.989
C03187=1073.657,-28.301,439.770,173.053,22.372,153.989
C03188=1073.651,-28.551,439.783,173.052,22.370,153.989
C03189=1073.645,-28.800,439.796,173.050,22.368,153.989
C03190=1073.639,-29.050,439.809,173.049,22.365,153.988
C03191=1073.633,-29.299,439.822,173.048,22.363,153.988
C03192=1073.627,-29.549,439.835,173.046,22.361,153.988
C03193=1073.621,-29.798,439.848,173.044,22.359,153.988
C03194=1073.615,-30.048,439.860,173.043,22.357,153.988
C03195=1073.610,-30.298,439.874,173.041,22.354,153.987
C03196=1073.604,-30.548,439.887,173.040,22.352,153.987
C03197=1073.598,-30.798,439.899,173.039,22.350,153.987
C03198=1073.592,-31.047,439.913,173.037,22.348,153.987
C03199=1073.586,-31.297,439.925,173.036,22.345,153.986
C03200=1073.580,-31.547,439.938,173.035,22.343,153.986
C03201=1073.573,-31.795,439.950,173.033,22.342,153.986
C03202=1073.567,-32.045,439.963,173.031,22.339,153.986
C03203=1073.561,-32.295,439.976,173.030,22.337,153.986
C03204=1073.555,-32.545,439.989,173.029,22.334,153.985
C03205=1073.549,-32.794,440.001,173.027,22.332,153.985
C03206=1073.543,-33.043,440.014,173.026,22.330,153.985
C03207=1073.537,-33.319,440.029,173.025,22.328,153.985
C03208=1073.530,-33.595,440.042,173.022,22.325,153.985
C03209=1073.524,-33.870,440.056,173.021,22.323,153.984
C03210=1073.517,-34.146,440.070,173.020,22.321,153.984
C03211=1073.511,-34.396,440.083,173.019,22.318,153.984
C03212=1073.505,-34.645,440.096,173.016,22.316,153.984
C03213=1073.499,-34.895,440.108,173.015,22.314,153.983
C03214=1073.493,-35.145,440.121,173.014,22.312,153.983
C03215=1073.487,-35.394,440.134,173.012,22.310,153.983
C03216=1073.481,-35.644,440.147,173.011,22.307,153.983
C03217=1073.475,-35.894,440.159,173.010,22.305,153.983
C03218=1073.470,-36.143,440.171,173.008,22.303,153.982
C03219=1073.464,-36.392,440.185,173.007,22.301,153.982
C03220=1073.458,-36.642,440.197,173.006,22.299,153.982
C03221=1073.452,-36.892,440.210,173.004,22.297,153.982
C03222=1073.446,-37.142,440.222,173.002,22.294,153.982
C03223=1073.440,-37.391,440.236,173.001,22.292,153.982
C03224=1073.434,-37.641,440.248,173.000,22.290,153.981
C03225=1073.428,-37.890,440.260,172.998,22.288,153.981
C03226=1073.422,-38.140,440.272,172.997,22.285,153.981
C03227=1073.416,-38.390,440.285,172.995,22.284,153.981
C03228=1073.410,-38.639,440.298,172.994,22.282,153.981
C03229=1073.404,-38.889,440.311,172.993,22.279,153.980
C03230=1073.398,-39.139,440.323,172.991,22.277,153.980
C03231=1073.393,-39.388,440.336,172.989,22.275,153.980
C03232=1073.386,-39.637,440.347,172.988,22.273,153.980
C03233=1073.380,-39.887,440.360,172.987,22.271,153.980
C03234=1073.374,-40.137,440.373,172.985,22.269,153.979
C03235=1073.368,-40.386,440.386,172.984,22.267,153.979
C03236=1073.361,-40.636,440.398,172.982,22.265,153.979
C03237=1073.355,-40.886,440.410,172.981,22.262,153.979
C03238=1073.350,-41.135,440.423,172.980,22.260,153.979
C03239=1073.343,-41.385,440.435,172.978,22.258,153.979
C03240=1073.337,-41.634,440.447,172.977,22.257,153.978
C03241=1073.332,-41.884,440.460,172.976,22.254,153.978
C03242=1073.326,-42.134,440.472,172.973,22.252,153.978
C03243=1073.319,-42.384,440.484,172.972,22.250,153.978
C03244=1073.314,-42.633,440.496,172.971,22.248,153.978
C03245=1073.308,-42.883,440.509,172.969,22.245,153.977
C03246=1073.301,-43.132,440.521,172.968,22.244,153.977
C03247=1073.295,-43.382,440.533,172.967,22.242,153.977
C03248=1073.289,-43.632,440.546,172.965,22.240,153.977
C03249=1073.284,-43.881,440.558,172.964,22.237,153.977
C03250=1073.277,-44.130,440.571,172.963,22.235,153.976
C03251=1073.271,-44.380,440.583,172.961,22.233,153.976
C03252=1073.265,-44.630,440.596,172.959,22.231,153.976
C03253=1073.259,-44.879,440.608,172.957,22.229,153.976
C03254=1073.254,-45.129,440.619,172.956,22.227,153.976
C03255=1073.248,-45.379,440.632,172.955,22.225,153.976
C03256=1073.241,-45.629,440.644,172.953,22.223,153.975
C03257=1073.236,-45.878,440.656,172.952,22.221,153.975
C03258=1073.230,-46.128,440.669,172.951,22.219,153.975
C03259=1073.223,-46.378,440.681,172.949,22.217,153.975
C03260=1073.217,-46.627,440.693,172.948,22.215,153.975
C03261=1073.212,-46.877,440.705,172.947,22.213,153.975
C03262=1073.205,-47.126,440.717,172.945,22.211,153.974
C03263=1073.199,-47.376,440.730,172.943,22.208,153.974
C03264=1073.194,-47.626,440.742,172.942,22.207,153.974
C03265=1073.187,-47.875,440.754,172.940,22.204,153.974
C03266=1073.182,-48.125,440.767,172.939,22.202,153.974
C03267=1073.176,-48.375,440.779,172.938,22.200,153.974
C03268=1073.170,-48.623,440.791,172.936,22.198,153.973
C03269=1073.164,-48.874,440.803,172.935,22.196,153.973
C03270=1073.157,-49.124,440.814,172.933,22.194,153.973
C03271=1073.151,-49.399,440.829,172.932,22.192,153.973
C03272=1073.145,-49.675,440.841,172.930,22.190,153.973
C03273=1073.138,-49.951,440.855,172.929,22.187,153.972
C03274=1073.131,-50.227,440.868,172.927,22.185,153.972
C03275=1073.125,-50.477,440.881,172.925,22.183,153.972
C03276=1073.119,-50.726,440.892,172.924,22.181,153.972
C03277=1073.114,-50.976,440.904,172.922,22.179,153.972
C03278=1073.107,-51.226,440.916,172.921,22.177,153.972
C03279=1073.101,-51.476,440.929,172.919,22.175,153.972
C03280=1073.095,-51.725,440.940,172.918,22.173,153.971
C03281=1073.088,-51.974,440.952,172.917,22.171,153.971
C03282=1073.083,-52.225,440.964,172.915,22.169,153.971
C03283=1073.076,-52.474,440.976,172.914,22.168,153.971
C03284=1073.070,-52.723,440.988,172.912,22.166,153.971
C03285=1073.064,-52.973,441.000,172.911,22.164,153.971
C03286=1073.058,-53.223,441.011,172.910,22.162,153.971
C03287=1073.052,-53.472,441.023,172.908,22.160,153.970
C03288=1073.046,-53.722,441.036,172.906,22.158,153.970
C03289=1073.039,-53.972,441.048,172.905,22.156,153.970
C03290=1073.033,-54.222,441.059,172.903,22.154,153.970
C03291=1073.027,-54.471,441.071,172.902,22.152,153.970
C03292=1073.021,-54.721,441.083,172.900,22.150,153.970
C03293=1073.014,-54.971,441.094,172.899,22.148,153.970
C03294=1073.009,-55.220,441.106,172.897,22.147,153.969
C03295=1073.003,-55.470,441.118,172.896,22.145,153.969
C03296=1072.996,-55.720,441.130,172.895,22.143,153.969
C03297=1072.991,-55.969,441.142,172.893,22.141,153.969
C03298=1072.984,-56.219,441.154,172.892,22.139,153.969
C03299=1072.978,-56.469,441.165,172.890,22.137,153.969
C03300=1072.973,-56.718,441.177,172.889,22.135,153.969
C03301=1072.966,-56.967,441.189,172.887,22.133,153.968
C03302=1072.960,-57.218,441.200,172.885,22.131,153.968
C03303=1072.954,-57.467,441.213,172.884,22.129,153.968
C03304=1072.948,-57.716,441.224,172.882,22.127,153.968
C03305=1072.941,-57.967,441.236,172.881,22.126,153.968
C03306=1072.936,-58.216,441.248,172.880,22.124,153.968
C03307=1072.930,-58.466,441.259,172.878,22.122,153.968
C03308=1072.924,-58.715,441.271,172.877,22.120,153.968
C03309=1072.917,-58.964,441.283,172.875,22.118,153.967
C03310=1072.911,-59.215,441.295,172.874,22.116,153.967
C03311=1072.905,-59.464,441.306,172.873,22.114,153.967
C03312=1072.899,-59.714,441.317,172.871,22.113,153.967
C03313=1072.893,-59.963,441.329,172.870,22.111,153.967
C03314=1072.887,-60.213,441.341,172.868,22.109,153.967
C03315=1072.881,-60.463,441.353,172.866,22.106,153.967
C03316=1072.875,-60.712,441.364,172.864,22.104,153.966
C03317=1072.869,-60.962,441.376,172.863,22.103,153.966
C03318=1072.863,-61.211,441.388,172.862,22.101,153.966
C03319=1072.857,-61.461,441.399,172.860,22.099,153.966
C03320=1072.850,-61.711,441.411,172.859,22.097,153.966
C03321=1072.845,-61.961,441.422,172.857,22.095,153.966
C03322=1072.838,-62.210,441.434,172.856,22.093,153.966
C03323=1072.833,-62.460,441.445,172.855,22.092,153.966
C03324=1072.826,-62.710,441.457,172.853,22.090,153.965
C03325=1072.821,-62.959,441.469,172.852,22.088,153.965
C03326=1072.815,-63.209,441.480,172.850,22.086,153.965
C03327=1072.809,-63.458,441.492,172.849,22.084,153.965
C03328=1072.802,-63.708,441.503,172.847,22.082,153.965
C03329=1072.797,-63.958,441.515,172.846,22.081,153.965
C03330=1072.791,-64.208,441.526,172.843,22.079,153.965
C03331=1072.785,-64.457,441.538,172.842,22.077,153.965
C03332=1072.778,-64.707,441.549,172.841,22.075,153.965
C03333=1072.772,-64.956,441.560,172.839,22.073,153.964
C03334=1072.767,-65.206,441.573,172.838,22.071,153.964
C03335=1072.760,-65.484,441.585,172.837,22.069,153.964
C03336=1072.753,-65.761,441.598,172.835,22.067,153.964
C03337=1072.746,-66.038,441.610,172.833,22.065,153.964
C03338=1072.740,-66.315,441.622,172.831,22.063,153.964
C03339=1072.734,-66.565,441.635,172.830,22.062,153.964
C03340=1072.728,-66.815,441.646,172.828,22.060,153.963
C03341=1072.722,-67.064,441.657,172.827,22.058,153.963
C03342=1072.716,-67.314,441.669,172.826,22.056,153.963
C03343=1072.710,-67.563,441.680,172.824,22.054,153.963
C03344=1072.704,-67.814,441.691,172.823,22.052,153.963
C03345=1072.698,-68.063,441.703,172.821,22.051,153.963
C03346=1072.692,-68.313,441.714,172.820,22.049,153.963
C03347=1072.686,-68.562,441.725,172.818,22.047,153.963
C03348=1072.679,-68.812,441.737,172.817,22.045,153.963
C03349=1072.674,-69.062,441.749,172.815,22.043,153.962
C03350=1072.669,-69.311,441.759,172.813,22.042,153.962
C03351=1072.662,-69.561,441.771,172.812,22.040,153.962
C03352=1072.656,-69.810,441.782,172.810,22.038,153.962
C03353=1072.650,-70.061,441.794,172.809,22.036,153.962
C03354=1072.644,-70.310,441.804,172.807,22.034,153.962
C03355=1072.638,-70.560,441.816,172.806,22.032,153.962
C03356=1072.633,-70.809,441.828,172.805,22.031,153.962
C03357=1072.627,-71.059,441.839,172.803,22.029,153.962
C03358=1072.620,-71.309,441.850,172.802,22.027,153.961
C03359=1072.615,-71.559,441.861,172.800,22.025,153.961
C03360=1072.608,-71.808,441.873,172.799,22.024,153.961
C03361=1072.602,-72.058,441.884,172.797,22.022,153.961
C03362=1072.597,-72.307,441.895,172.796,22.020,153.961
C03363=1072.591,-72.558,441.906,172.794,22.019,153.961
C03364=1072.585,-72.807,441.917,172.793,22.017,153.961
C03365=1072.579,-73.056,441.929,172.791,22.015,153.961
C03366=1072.573,-73.306,441.940,172.790,22.013,153.961
C03367=1072.567,-73.556,441.951,172.788,22.012,153.961
C03368=1072.561,-73.805,441.962,172.787,22.010,153.960
C03369=1072.555,-74.055,441.973,172.786,22.008,153.960
C03370=1072.549,-74.305,441.984,172.783,22.006,153.960
C03371=1072.543,-74.554,441.996,172.782,22.005,153.960
C03372=1072.537,-74.804,442.007,172.780,22.003,153.960
C03373=1072.531,-75.053,442.018,172.779,22.001,153.960
C03374=1072.525,-75.304,442.029,172.777,21.999,153.960
C03375=1072.519,-75.553,442.040,172.776,21.998,153.960
C03376=1072.513,-75.803,442.051,172.774,21.996,153.960
C03377=1072.507,-76.053,442.062,172.773,21.995,153.960
C03378=1072.501,-76.302,442.073,172.771,21.993,153.960
C03379=1072.495,-76.552,442.084,172.770,21.991,153.960
C03380=1072.489,-76.802,442.094,172.768,21.989,153.959
C03381=1072.482,-77.052,442.106,172.767,21.988,153.959
C03382=1072.476,-77.301,442.117,172.765,21.986,153.959
C03383=1072.470,-77.550,442.128,172.764,21.985,153.959
C03384=1072.464,-77.800,442.139,172.762,21.983,153.959
C03385=1072.458,-78.050,442.150,172.761,21.981,153.959
C03386=1072.453,-78.299,442.161,172.759,21.979,153.959
C03387=1072.446,-78.550,442.172,172.758,21.978,153.959
C03388=1072.440,-78.799,442.183,172.756,21.976,153.959
C03389=1072.435,-79.049,442.194,172.755,21.975,153.959
C03390=1072.428,-79.298,442.205,172.753,21.973,153.959
C03391=1072.422,-79.548,442.216,172.752,21.971,153.959
C03392=1072.416,-79.797,442.226,172.750,21.970,153.959
C03393=1072.410,-80.048,442.238,172.749,21.968,153.958
C03394=1072.404,-80.297,442.249,172.747,21.967,153.958
C03395=1072.398,-80.546,442.259,172.746,21.965,153.958
C03396=1072.391,-80.796,442.270,172.744,21.963,153.958
C03397=1072.386,-81.046,442.281,172.743,21.962,153.958
C03398=1072.379,-81.296,442.291,172.741,21.961,153.958
C03399=1072.372,-81.575,442.304,172.739,21.958,153.958
C03400=1072.365,-81.855,442.315,172.737,21.957,153.958
C03401=1072.358,-82.134,442.328,172.736,21.955,153.958
C03402=1072.352,-82.414,442.340,172.734,21.954,153.958
C03403=1072.345,-82.664,442.350,172.733,21.952,153.958
C03404=1072.339,-82.913,442.361,172.730,21.950,153.958
C03405=1072.334,-83.163,442.372,172.729,21.949,153.958
C03406=1072.327,-83.413,442.382,172.727,21.947,153.958
C03407=1072.321,-83.663,442.393,172.726,21.946,153.958
C03408=1072.315,-83.912,442.404,172.724,21.944,153.958
C03409=1072.308,-84.162,442.414,172.723,21.942,153.958
C03410=1072.302,-84.411,442.425,172.721,21.941,153.957
C03411=1072.297,-84.661,442.436,172.720,21.940,153.957
C03412=1072.290,-84.911,442.447,172.718,21.938,153.957
C03413=1072.284,-85.161,442.457,172.717,21.936,153.957
C03414=1072.278,-85.410,442.468,172.715,21.935,153.957
C03415=1072.271,-85.660,442.478,172.714,21.934,153.957
C03416=1072.266,-85.910,442.489,172.712,21.932,153.957
C03417=1072.260,-86.159,442.500,172.711,21.930,153.957
C03418=1072.253,-86.408,442.510,172.709,21.929,153.957
C03419=1072.247,-86.659,442.521,172.707,21.928,153.957
C03420=1072.242,-86.909,442.532,172.706,21.926,153.957
C03421=1072.235,-87.158,442.542,172.704,21.925,153.957
C03422=1072.229,-87.407,442.553,172.703,21.923,153.957
C03423=1072.223,-87.658,442.563,172.701,21.921,153.957
C03424=1072.217,-87.907,442.574,172.700,21.920,153.957
C03425=1072.211,-88.157,442.585,172.698,21.919,153.957
C03426=1072.205,-88.406,442.595,172.697,21.917,153.957
C03427=1072.199,-88.657,442.606,172.695,21.916,153.957
C03428=1072.193,-88.906,442.616,172.694,21.914,153.957
C03429=1072.186,-89.156,442.627,172.692,21.913,153.957
C03430=1072.181,-89.405,442.638,172.690,21.911,153.957
C03431=1072.174,-89.655,442.648,172.689,21.910,153.957
C03432=1072.168,-89.905,442.658,172.687,21.908,153.957
C03433=1072.162,-90.154,442.669,172.686,21.907,153.957
C03434=1072.156,-90.404,442.679,172.684,21.906,153.957
C03435=1072.151,-90.654,442.690,172.683,21.904,153.956
C03436=1072.144,-90.904,442.700,172.681,21.902,153.956
C03437=1072.138,-91.154,442.711,172.680,21.901,153.956
C03438=1072.132,-91.403,442.721,172.678,21.900,153.956
C03439=1072.126,-91.652,442.732,172.676,21.898,153.956
C03440=1072.120,-91.903,442.742,172.675,21.897,153.956
C03441=1072.114,-92.152,442.752,172.673,21.895,153.956
C03442=1072.108,-92.402,442.763,172.672,21.894,153.956
C03443=1072.101,-92.652,442.773,172.670,21.893,153.956
C03444=1072.096,-92.901,442.784,172.669,21.891,153.956
C03445=1072.090,-93.151,442.794,172.667,21.889,153.956
C03446=1072.084,-93.400,442.804,172.666,21.888,153.956
C03447=1072.078,-93.650,442.815,172.664,21.887,153.956
C03448=1072.071,-93.900,442.825,172.662,21.885,153.956
C03449=1072.066,-94.150,442.836,172.661,21.884,153.956
C03450=1072.059,-94.400,442.846,172.659,21.882,153.956
C03451=1072.054,-94.649,442.856,172.658,21.881,153.956
C03452=1072.047,-94.899,442.866,172.656,21.880,153.956
C03453=1072.042,-95.149,442.877,172.655,21.878,153.956
C03454=1072.036,-95.398,442.888,172.653,21.877,153.956
C03455=1072.030,-95.648,442.897,172.651,21.876,153.956
C03456=1072.023,-95.898,442.909,172.650,21.874,153.956
C03457=1072.017,-96.148,442.918,172.648,21.873,153.956
C03458=1072.012,-96.397,442.929,172.647,21.871,153.956
C03459=1072.005,-96.647,442.939,172.645,21.870,153.956
C03460=1072.000,-96.897,442.949,172.643,21.869,153.956
C03461=1071.993,-97.146,442.959,172.642,21.867,153.956
C03462=1071.988,-97.396,442.970,172.640,21.866,153.956
C03463=1071.981,-97.678,442.981,172.639,21.865,153.956
C03464=1071.974,-97.959,442.993,172.637,21.863,153.956
C03465=1071.967,-98.242,443.004,172.636,21.862,153.956
C03466=1071.960,-98.523,443.016,172.634,21.860,153.956
C03467=1071.954,-98.773,443.026,172.632,21.859,153.956
C03468=1071.947,-99.022,443.036,172.631,21.858,153.956
C03469=1071.942,-99.272,443.046,172.629,21.856,153.956
C03470=1071.936,-99.522,443.056,172.627,21.855,153.956
C03471=1071.929,-99.771,443.066,172.626,21.854,153.956
C03472=1071.924,-100.022,443.076,172.624,21.853,153.956
C03473=1071.917,-100.271,443.087,172.623,21.851,153.956
C03474=1071.911,-100.521,443.096,172.621,21.850,153.956
C03475=1071.904,-100.770,443.107,172.620,21.848,153.956
C03476=1071.899,-101.021,443.117,172.618,21.848,153.956
C03477=1071.893,-101.270,443.126,172.616,21.846,153.956
C03478=1071.886,-101.520,443.137,172.615,21.845,153.956
C03479=1071.881,-101.770,443.147,172.613,21.843,153.956
C03480=1071.874,-102.019,443.157,172.611,21.842,153.956
C03481=1071.868,-102.269,443.167,172.610,21.841,153.956
C03482=1071.863,-102.519,443.177,172.608,21.840,153.956
C03483=1071.856,-102.768,443.187,172.607,21.839,153.956
C03484=1071.850,-103.018,443.197,172.605,21.837,153.956
C03485=1071.844,-103.267,443.206,172.603,21.836,153.956
C03486=1071.837,-103.518,443.217,172.602,21.835,153.956
C03487=1071.831,-103.767,443.227,172.600,21.834,153.956
C03488=1071.825,-104.017,443.236,172.598,21.832,153.956
C03489=1071.819,-104.267,443.247,172.597,21.831,153.956
C03490=1071.813,-104.517,443.257,172.595,21.830,153.956
C03491=1071.807,-104.766,443.267,172.594,21.829,153.956
C03492=1071.801,-105.016,443.276,172.592,21.827,153.956
C03493=1071.795,-105.266,443.287,172.590,21.826,153.956
C03494=1071.789,-105.515,443.297,172.589,21.825,153.956
C03495=1071.783,-105.765,443.306,172.588,21.824,153.956
C03496=1071.777,-106.015,443.316,172.586,21.823,153.956
C03497=1071.771,-106.265,443.327,172.585,21.822,153.956
C03498=1071.765,-106.514,443.336,172.583,21.820,153.956
C03499=1071.758,-106.764,443.346,172.581,21.820,153.956
C03500=1071.752,-107.014,443.355,172.580,21.818,153.956
C03501=1071.746,-107.263,443.366,172.578,21.817,153.956
C03502=1071.740,-107.513,443.376,172.576,21.816,153.956
C03503=1071.734,-107.763,443.385,172.575,21.815,153.956
C03504=1071.728,-108.013,443.395,172.573,21.814,153.956
C03505=1071.722,-108.263,443.404,172.571,21.812,153.956
C03506=1071.715,-108.512,443.415,172.570,21.811,153.956
C03507=1071.709,-108.762,443.424,172.568,21.810,153.956
C03508=1071.703,-109.011,443.434,172.566,21.809,153.956
C03509=1071.697,-109.261,443.443,172.565,21.808,153.957
C03510=1071.691,-109.511,443.454,172.563,21.807,153.957
C03511=1071.685,-109.761,443.463,172.561,21.806,153.957
C03512=1071.679,-110.010,443.473,172.560,21.804,153.957
C03513=1071.673,-110.260,443.483,172.558,21.803,153.957
C03514=1071.666,-110.510,443.492,172.556,21.802,153.957
C03515=1071.660,-110.760,443.502,172.556,21.801,153.957
C03516=1071.654,-111.009,443.512,172.554,21.800,153.957
C03517=1071.648,-111.259,443.521,172.552,21.799,153.957
C03518=1071.642,-111.509,443.531,172.551,21.798,153.957
C03519=1071.636,-111.759,443.540,172.549,21.797,153.957
C03520=1071.629,-112.008,443.551,172.547,21.796,153.957
C03521=1071.623,-112.258,443.560,172.546,21.795,153.957
C03522=1071.618,-112.508,443.570,172.544,21.794,153.957
C03523=1071.611,-112.758,443.580,172.542,21.792,153.957
C03524=1071.605,-113.008,443.589,172.541,21.791,153.957
C03525=1071.600,-113.257,443.599,172.539,21.790,153.957
C03526=1071.593,-113.506,443.608,172.537,21.789,153.957
C03527=1071.586,-113.786,443.618,172.536,21.788,153.957
C03528=1071.580,-114.065,443.630,172.534,21.787,153.957
C03529=1071.572,-114.345,443.640,172.532,21.786,153.957
C03530=1071.566,-114.624,443.651,172.530,21.785,153.957
C03531=1071.559,-114.874,443.661,172.529,21.784,153.958
C03532=1071.553,-115.124,443.670,172.527,21.783,153.958
C03533=1071.547,-115.374,443.680,172.525,21.782,153.958
C03534=1071.541,-115.623,443.690,172.524,21.780,153.958
C03535=1071.535,-115.872,443.699,172.522,21.780,153.958
C03536=1071.529,-116.122,443.708,172.520,21.779,153.958
C03537=1071.523,-116.372,443.718,172.519,21.777,153.958
C03538=1071.517,-116.622,443.727,172.517,21.777,153.958
C03539=1071.511,-116.872,443.737,172.515,21.776,153.958
C03540=1071.505,-117.121,443.747,172.514,21.774,153.958
C03541=1071.498,-117.371,443.756,172.513,21.774,153.958
C03542=1071.491,-117.621,443.765,172.511,21.773,153.958
C03543=1071.485,-117.871,443.775,172.509,21.772,153.958
C03544=1071.479,-118.121,443.784,172.508,21.771,153.958
C03545=1071.474,-118.370,443.793,172.506,21.770,153.959
C03546=1071.468,-118.620,443.802,172.504,21.769,153.959
C03547=1071.462,-118.870,443.812,172.502,21.768,153.959
C03548=1071.455,-119.119,443.821,172.501,21.767,153.959
C03549=1071.449,-119.369,443.831,172.499,21.766,153.959
C03550=1071.443,-119.619,443.841,172.497,21.765,153.959
C03551=1071.437,-119.869,443.850,172.495,21.764,153.959
C03552=1071.431,-120.119,443.860,172.494,21.763,153.959
C03553=1071.424,-120.367,443.868,172.493,21.763,153.959
C03554=1071.418,-120.618,443.877,172.491,21.761,153.959
C03555=1071.412,-120.868,443.887,172.489,21.761,153.959
C03556=1071.406,-121.117,443.896,172.488,21.760,153.959
C03557=1071.400,-121.367,443.906,172.486,21.759,153.959
C03558=1071.394,-121.617,443.915,172.484,21.758,153.960
C03559=1071.388,-121.867,443.925,172.483,21.757,153.960
C03560=1071.382,-122.116,443.933,172.481,21.756,153.960
C03561=1071.375,-122.366,443.942,172.479,21.755,153.960
C03562=1071.369,-122.616,443.952,172.477,21.754,153.960
C03563=1071.363,-122.866,443.962,172.476,21.754,153.960
C03564=1071.357,-123.115,443.971,172.475,21.752,153.960
C03565=1071.351,-123.366,443.980,172.473,21.752,153.960
C03566=1071.345,-123.615,443.989,172.471,21.751,153.960
C03567=1071.339,-123.864,443.998,172.469,21.750,153.960
C03568=1071.332,-124.114,444.008,172.468,21.749,153.960
C03569=1071.327,-124.365,444.017,172.466,21.748,153.961
C03570=1071.320,-124.614,444.026,172.464,21.747,153.961
C03571=1071.314,-124.863,444.035,172.463,21.746,153.961
C03572=1071.308,-125.113,444.044,172.461,21.745,153.961
C03573=1071.302,-125.363,444.053,172.460,21.745,153.961
C03574=1071.296,-125.613,444.063,172.458,21.744,153.961
C03575=1071.289,-125.863,444.072,172.456,21.743,153.961
C03576=1071.283,-126.112,444.081,172.455,21.742,153.961
C03577=1071.278,-126.362,444.090,172.453,21.741,153.961
C03578=1071.271,-126.612,444.099,172.451,21.741,153.961
C03579=1071.264,-126.861,444.108,172.449,21.740,153.962
C03580=1071.259,-127.112,444.117,172.447,21.739,153.962
C03581=1071.252,-127.362,444.127,172.446,21.738,153.962
C03582=1071.246,-127.610,444.135,172.445,21.738,153.962
C03583=1071.240,-127.862,444.145,172.443,21.737,153.962
C03584=1071.235,-128.113,444.155,172.441,21.736,153.962
C03585=1071.232,-128.363,444.165,172.440,21.734,153.962
C03586=1071.231,-128.614,444.176,172.439,21.731,153.962
C03587=1071.232,-128.867,444.189,172.438,21.727,153.961
C03588=1071.236,-129.120,444.201,172.438,21.723,153.960
C03589=1071.241,-129.372,444.216,172.437,21.718,153.960
C03590=1071.248,-129.622,444.230,172.437,21.713,153.959
C03591=1070.858,-129.644,444.066,172.390,21.851,153.991
C03592=1070.850,-129.394,444.051,172.390,21.857,153.992
C03593=1070.845,-129.143,444.038,172.391,21.861,153.992
C03594=1070.841,-128.889,444.024,172.391,21.866,153.993
C03595=1070.840,-128.636,444.012,172.392,21.869,153.994
C03596=1070.841,-128.386,444.001,172.393,21.872,153.994
C03597=1070.844,-128.135,443.990,172.395,21.874,153.994
C03598=1070.848,-127.884,443.980,172.396,21.875,153.994
C03599=1070.854,-127.633,443.971,172.398,21.876,153.994
C03600=1070.860,-127.384,443.962,172.400,21.877,153.994
C03601=1070.867,-127.134,443.953,172.402,21.878,153.994
C03602=1070.873,-126.884,443.944,172.404,21.878,153.994
C03603=1070.879,-126.634,443.935,172.405,21.879,153.994
C03604=1070.886,-126.385,443.926,172.406,21.880,153.993
C03605=1070.892,-126.135,443.916,172.408,21.880,153.993
C03606=1070.898,-125.885,443.908,172.410,21.881,153.993
C03607=1070.904,-125.635,443.898,172.412,21.882,153.993
C03608=1070.911,-125.386,443.889,172.413,21.883,153.993
C03609=1070.916,-125.136,443.880,172.415,21.884,153.993
C03610=1070.922,-124.886,443.871,172.417,21.885,153.993
C03611=1070.928,-124.636,443.861,172.418,21.886,153.993
C03612=1070.935,-124.387,443.852,172.420,21.887,153.993
C03613=1070.941,-124.136,443.844,172.421,21.887,153.993
C03614=1070.947,-123.887,443.834,172.423,21.888,153.992
C03615=1070.953,-123.637,443.825,172.425,21.889,153.992
C03616=1070.959,-123.388,443.815,172.426,21.890,153.992
C03617=1070.966,-123.138,443.806,172.428,21.890,153.992
C03618=1070.972,-122.888,443.797,172.430,21.892,153.992
C03619=1070.978,-122.638,443.788,172.432,21.893,153.992
C03620=1070.984,-122.388,443.778,172.433,21.893,153.992
C03621=1070.990,-122.139,443.769,172.435,21.894,153.992
C03622=1070.996,-121.889,443.759,172.437,21.895,153.992
C03623=1071.002,-121.639,443.751,172.438,21.896,153.992
C03624=1071.009,-121.389,443.742,172.439,21.897,153.992
C03625=1071.015,-121.140,443.732,172.441,21.898,153.991
C03626=1071.021,-120.890,443.723,172.443,21.899,153.991
C03627=1071.027,-120.641,443.713,172.444,21.900,153.991
C03628=1071.033,-120.391,443.704,172.446,21.901,153.991
C03629=1071.039,-120.140,443.695,172.448,21.902,153.991
C03630=1071.045,-119.891,443.685,172.450,21.902,153.991
C03631=1071.051,-119.641,443.676,172.451,21.904,153.991
C03632=1071.058,-119.391,443.667,172.453,21.905,153.991
